            FOR i := 1 TO 10 DO
                GVL_1.Condition_Cr_A[condNo].Row[i].Enable   := GVL.HMI_A_CondEditRowEnable[i];
                GVL_1.Condition_Cr_A[condNo].Row[i].Source   := GVL.HMI_A_CondEditSource[i];
                GVL_1.Condition_Cr_A[condNo].Row[i].Index    := GVL.HMI_A_CondEditIndex[i];
                GVL_1.Condition_Cr_A[condNo].Row[i].Operator := GVL.HMI_A_CondEditOperator[i];
                GVL_1.Condition_Cr_A[condNo].Row[i].SetValue := GVL.HMI_A_CondEditSetValue[i];
                GVL_1.Condition_Cr_A[condNo].Row[i].LinkNext := GVL.HMI_A_CondEditLinkNext[i];
                //GVL_1.Condition_Cr_A[condNo].Row[i].Note     := GVL.HMI_A_CondEditNote[i];
            END_FOR;
        END_IF;

        GVL.HMI_A_CondCmdReq := 0;


    3: // Clear condition
        condNo := GVL.HMI_A_CondSelectedNo;

        IF (condNo >= 1) AND (condNo <= 100) THEN
            GVL_1.Condition_Cr_A[condNo].Enable := FALSE;
            GVL_1.Condition_Cr_A[condNo].Name := '';

            FOR i := 1 TO 10 DO
                GVL_1.Condition_Cr_A[condNo].Row[i].Enable := FALSE;
                GVL_1.Condition_Cr_A[condNo].Row[i].Source := 0;
                GVL_1.Condition_Cr_A[condNo].Row[i].Index := 0;
                GVL_1.Condition_Cr_A[condNo].Row[i].Operator := 0;
                GVL_1.Condition_Cr_A[condNo].Row[i].SetValue := 0;
                GVL_1.Condition_Cr_A[condNo].Row[i].LinkNext := 0;
                //GVL_1.Condition_Cr_A[condNo].Row[i].Note := '';
            END_FOR;
        END_IF;

        GVL.HMI_A_CondCmdReq := 0;


    4: // Copy
        condNo := GVL.HMI_A_CondSelectedNo;

        IF (condNo >= 1) AND (condNo <= 100) THEN
            GVL.HMI_A_CondCopied := GVL_1.Condition_Cr_A[condNo];
        END_IF;

        GVL.HMI_A_CondCmdReq := 0;


    5: // Paste
        condNo := GVL.HMI_A_CondEditNo;

        IF (condNo >= 1) AND (condNo <= 100) THEN
            GVL_1.Condition_Cr_A[condNo] := GVL.HMI_A_CondCopied;
        END_IF;

        GVL.HMI_A_CondCmdReq := 1; // Load lại lên Edit


    6: // Delete Row
        rowNo := GVL.HMI_A_CondSelectedNo;

        IF (rowNo >= 1) AND (rowNo <= 10) THEN
            FOR i := rowNo TO 9 DO
                GVL.HMI_A_CondEditRowEnable[i] := GVL.HMI_A_CondEditRowEnable[i + 1];
                GVL.HMI_A_CondEditSource[i]    := GVL.HMI_A_CondEditSource[i + 1];
                GVL.HMI_A_CondEditIndex[i]     := GVL.HMI_A_CondEditIndex[i + 1];
                GVL.HMI_A_CondEditOperator[i]  := GVL.HMI_A_CondEditOperator[i + 1];
                GVL.HMI_A_CondEditSetValue[i]  := GVL.HMI_A_CondEditSetValue[i + 1];
                GVL.HMI_A_CondEditLinkNext[i]  := GVL.HMI_A_CondEditLinkNext[i + 1];
                GVL.HMI_A_CondEditNote[i]      := GVL.HMI_A_CondEditNote[i + 1];
            END_FOR;

            GVL.HMI_A_CondEditRowEnable[10] := FALSE;
            GVL.HMI_A_CondEditSource[10] := 0;
            GVL.HMI_A_CondEditIndex[10] := 0;
            GVL.HMI_A_CondEditOperator[10] := 0;
            GVL.HMI_A_CondEditSetValue[10] := 0;
            GVL.HMI_A_CondEditLinkNext[10] := 0;
            GVL.HMI_A_CondEditNote[10] := '';
        END_IF;

        GVL.HMI_A_CondCmdReq := 0;


    7: // Insert Row
        rowNo := GVL.HMI_A_CondSelectedNo;

        IF (rowNo >= 1) AND (rowNo <= 10) THEN
            FOR i := 10 TO rowNo + 1 BY -1 DO
                GVL.HMI_A_CondEditRowEnable[i] := GVL.HMI_A_CondEditRowEnable[i - 1];
                GVL.HMI_A_CondEditSource[i]    := GVL.HMI_A_CondEditSource[i - 1];
                GVL.HMI_A_CondEditIndex[i]     := GVL.HMI_A_CondEditIndex[i - 1];
                GVL.HMI_A_CondEditOperator[i]  := GVL.HMI_A_CondEditOperator[i - 1];
                GVL.HMI_A_CondEditSetValue[i]  := GVL.HMI_A_CondEditSetValue[i - 1];
                GVL.HMI_A_CondEditLinkNext[i]  := GVL.HMI_A_CondEditLinkNext[i - 1];
                GVL.HMI_A_CondEditNote[i]      := GVL.HMI_A_CondEditNote[i - 1];
            END_FOR;

            GVL.HMI_A_CondEditRowEnable[rowNo] := FALSE;
            GVL.HMI_A_CondEditSource[rowNo] := 0;
            GVL.HMI_A_CondEditIndex[rowNo] := 0;
            GVL.HMI_A_CondEditOperator[rowNo] := 0;
            GVL.HMI_A_CondEditSetValue[rowNo] := 0;
            GVL.HMI_A_CondEditLinkNext[rowNo] := 0;
            GVL.HMI_A_CondEditNote[rowNo] := '';
        END_IF;

        GVL.HMI_A_CondCmdReq := 0;

END_CASE;


// PRG_A_ConditionScan -- PRG quét realtime kết quả Condition
FOR i := 1 TO 100 DO
    GVL_1.Condition_Cr_A[i].Result := F_EvalCondition_A(i);
END_FOR;

//====================================================
// CONDITION EDIT MONITOR
// Khi bật Monitor, hiển thị ActualValue / RowResult / FinalResult
// theo vùng đang edit, kể cả chưa Save
//====================================================

IF GVL.HMI_A_CondMonitorEnable THEN

    firstRow := TRUE;
    finalResult := FALSE;

    FOR i := 1 TO 10 DO

        IF GVL.HMI_A_CondEditRowEnable[i] THEN

            rowResult := F_EvalCondRowFromEdit_A(i);

            GVL.HMI_A_CondMonRowResult[i] := rowResult;

            IF firstRow THEN
                finalResult := rowResult;
                firstRow := FALSE;
            ELSE
                CASE GVL.HMI_A_CondEditLinkNext[i - 1] OF
                    1: finalResult := finalResult AND rowResult;
                    2: finalResult := finalResult OR rowResult;
                ELSE
                    finalResult := finalResult AND rowResult;
                END_CASE;
            END_IF;

        ELSE
            GVL.HMI_A_CondMonActualValue[i] := 0;
            GVL.HMI_A_CondMonRowResult[i] := FALSE;
        END_IF;

    END_FOR;

    GVL.HMI_A_CondMonFinalResult := finalResult;

ELSE
    GVL.HMI_A_CondMonFinalResult := FALSE;

    FOR i := 1 TO 10 DO
        GVL.HMI_A_CondMonActualValue[i] := 0;
        GVL.HMI_A_CondMonRowResult[i] := FALSE;
    END_FOR;
END_IF;
END_ACTION

ACTION ACT_HMI_A_Vision_Tracking_Config:
//=============================================================================
// ACT_HMI_A_Vision_Tracking_Config
//-----------------------------------------------------------------------------
// HMI editor cho Vision Tracking Source Robot A.
// Pattern giống Sensor Source:
// Index -> Edit Struct -> Load / Save.
//=============================================================================


//=============================================================================
// 01. KIỂM TRA INDEX
//=============================================================================
IF GVL.g_uiHMIVisionSourceIndexA = 0
OR GVL.g_uiHMIVisionSourceIndexA > GVL.C_MAX_VISION_CHANNELS THEN
    GVL.g_uiHMIVisionSourceIndexA := 1;
END_IF;


//=============================================================================
// 02. LOAD SOURCE -> HMI BUFFER
//=============================================================================
IF GVL.g_xHMILoadVisionSourceA THEN

    GVL.g_stHMIVisionSourceA :=
        GVL.g_aVisionTrackingSourceConfigA[
            GVL.g_uiHMIVisionSourceIndexA
        ];

    GVL.g_xHMILoadVisionSourceA := FALSE;

END_IF;


//=============================================================================
// 03. SAVE HMI BUFFER -> SOURCE
//=============================================================================
IF GVL.g_xHMISaveVisionSourceA THEN

    GVL.g_aVisionTrackingSourceConfigA[
        GVL.g_uiHMIVisionSourceIndexA
    ] := GVL.g_stHMIVisionSourceA;

    GVL.g_xHMISaveVisionSourceA := FALSE;

    // Yêu cầu lưu toàn bộ Vision Source xuống file.
    GVL.g_xHMISaveAllVisionSourceA := TRUE;

END_IF;
END_ACTION

ACTION ACT_HMI_B_ConditionEditor:
//====================================================
// PRG_HMI_A_ConditionEditor
// Hiển thị danh sách condition + xử lý Load/Save/Edit
//====================================================

// Scroll danh sách condition
IF GVL.HMI_B_CondCmd_Up THEN
    GVL.HMI_B_CondCmd_Up := FALSE;
    IF GVL.HMI_B_CondViewStart > 1 THEN
        GVL.HMI_B_CondViewStart := GVL.HMI_B_CondViewStart - 1;
    END_IF;
END_IF;

IF GVL.HMI_B_CondCmd_Down THEN
    GVL.HMI_B_CondCmd_Down := FALSE;
    IF GVL.HMI_B_CondViewStart < 91 THEN
        GVL.HMI_B_CondViewStart := GVL.HMI_B_CondViewStart + 1;
    END_IF;
END_IF;

IF GVL.HMI_B_CondCmd_PageUp THEN
    GVL.HMI_B_CondCmd_PageUp := FALSE;
    GVL.HMI_B_CondViewStart := GVL.HMI_B_CondViewStart - 10;
    IF GVL.HMI_B_CondViewStart < 1 THEN
        GVL.HMI_B_CondViewStart := 1;
    END_IF;
END_IF;

IF GVL.HMI_B_CondCmd_PageDown THEN
    GVL.HMI_B_CondCmd_PageDown := FALSE;
    GVL.HMI_B_CondViewStart := GVL.HMI_B_CondViewStart + 10;
    IF GVL.HMI_B_CondViewStart > 91 THEN
        GVL.HMI_B_CondViewStart := 91;
    END_IF;
END_IF;

IF GVL.HMI_B_CondCmd_GoTop THEN
    GVL.HMI_B_CondCmd_GoTop := FALSE;
    GVL.HMI_B_CondViewStart := 1;
END_IF;

IF GVL.HMI_B_CondCmd_GoBot THEN
    GVL.HMI_B_CondCmd_GoBot := FALSE;
    GVL.HMI_B_CondViewStart := 91;
END_IF;


//====================================================
// Row Select
//====================================================

FOR i := 1 TO 10 DO
    IF (GVL.HMI_B_CondSelectedCmd = i) THEN
		GVL.HMI_B_CondRowSelect[i] := TRUE;
		GVL.HMI_B_CondSelectedNo := i + GVL.HMI_B_CondViewStart - 1;
		//GVL.HMI_B_EditStepNo   := GVL.HMI_B_SelectedStepNo;
	ELSE
		GVL.HMI_B_CondRowSelect[i] := FALSE;
    END_IF;
END_FOR;

// FOR i := 1 TO 10 DO
//     IF GVL.HMI_B_CondRowSelect[i] THEN
//         GVL.HMI_B_CondRowSelect[i] := FALSE;
//         condNo := GVL.HMI_B_CondViewNo[i];
// 
//         IF (condNo >= 1) AND (condNo <= 100) THEN
//             GVL.HMI_B_CondSelectedNo := condNo;
//             GVL.HMI_B_CondCmdReq := 1; // Load
//         END_IF;
//     END_IF;
// END_FOR;


//====================================================
// Update View 10 dòng condition
//====================================================
FOR i := 1 TO 10 DO
    condNo := GVL.HMI_B_CondViewStart + i - 1;

    IF (condNo >= 1) AND (condNo <= 100) THEN
        GVL.HMI_B_CondViewNo[i]     := condNo;
        GVL.HMI_B_CondViewName[i]   := GVL_1.Condition_Cr_B[condNo].Name;
        GVL.HMI_B_CondViewEnable[i] := GVL_1.Condition_Cr_B[condNo].Enable;
        GVL.HMI_B_CondViewResult[i] := GVL_1.Condition_Cr_B[condNo].Result;
    ELSE
        GVL.HMI_B_CondViewNo[i]     := 0;
        GVL.HMI_B_CondViewName[i]   := '';
        GVL.HMI_B_CondViewEnable[i] := FALSE;
        GVL.HMI_B_CondViewResult[i] := FALSE;
    END_IF;
END_FOR;


//====================================================
// Command Load / Save / Clear / Copy / Paste
//====================================================
CASE GVL.HMI_B_CondCmdReq OF

    1: // Load condition vào vùng Edit
        condNo := GVL.HMI_B_CondSelectedNo;

        IF (condNo >= 1) AND (condNo <= 100) THEN
            GVL.HMI_B_CondEditNo := condNo;
            GVL.HMI_B_CondEditName := GVL_1.Condition_Cr_B[condNo].Name;
            GVL.HMI_B_CondEditEnable := GVL_1.Condition_Cr_B[condNo].Enable;

            FOR i := 1 TO 10 DO
                GVL.HMI_B_CondEditRowEnable[i] := GVL_1.Condition_Cr_B[condNo].Row[i].Enable;
                GVL.HMI_B_CondEditSource[i]    := GVL_1.Condition_Cr_B[condNo].Row[i].Source;
                GVL.HMI_B_CondEditIndex[i]     := GVL_1.Condition_Cr_B[condNo].Row[i].Index;
                GVL.HMI_B_CondEditOperator[i]  := GVL_1.Condition_Cr_B[condNo].Row[i].Operator;
                GVL.HMI_B_CondEditSetValue[i]  := GVL_1.Condition_Cr_B[condNo].Row[i].SetValue;
                GVL.HMI_B_CondEditLinkNext[i]  := GVL_1.Condition_Cr_B[condNo].Row[i].LinkNext;
                //GVL.HMI_B_CondEditNote[i]      := GVL_1.Condition_Cr_B[condNo].Row[i].Note;
            END_FOR;
        END_IF;

        GVL.HMI_B_CondCmdReq := 0;


    2: // Save vùng Edit về bảng thật
        condNo := GVL.HMI_B_CondSelectedNo;

        IF (condNo >= 1) AND (condNo <= 100) THEN
            GVL_1.Condition_Cr_B[condNo].Name := GVL.HMI_B_CondEditName;
            GVL_1.Condition_Cr_B[condNo].Enable := GVL.HMI_B_CondEditEnable;

            FOR i := 1 TO 10 DO
                GVL_1.Condition_Cr_B[condNo].Row[i].Enable   := GVL.HMI_B_CondEditRowEnable[i];
                GVL_1.Condition_Cr_B[condNo].Row[i].Source   := GVL.HMI_B_CondEditSource[i];
                GVL_1.Condition_Cr_B[condNo].Row[i].Index    := GVL.HMI_B_CondEditIndex[i];
                GVL_1.Condition_Cr_B[condNo].Row[i].Operator := GVL.HMI_B_CondEditOperator[i];
                GVL_1.Condition_Cr_B[condNo].Row[i].SetValue := GVL.HMI_B_CondEditSetValue[i];
                GVL_1.Condition_Cr_B[condNo].Row[i].LinkNext := GVL.HMI_B_CondEditLinkNext[i];
                //GVL_1.Condition_Cr_B[condNo].Row[i].Note     := GVL.HMI_B_CondEditNote[i];
            END_FOR;
        END_IF;

        GVL.HMI_B_CondCmdReq := 0;


    3: // Clear condition
        condNo := GVL.HMI_B_CondSelectedNo;

        IF (condNo >= 1) AND (condNo <= 100) THEN
            GVL_1.Condition_Cr_B[condNo].Enable := FALSE;
            GVL_1.Condition_Cr_B[condNo].Name := '';

            FOR i := 1 TO 10 DO
                GVL_1.Condition_Cr_B[condNo].Row[i].Enable := FALSE;
                GVL_1.Condition_Cr_B[condNo].Row[i].Source := 0;
                GVL_1.Condition_Cr_B[condNo].Row[i].Index := 0;
                GVL_1.Condition_Cr_B[condNo].Row[i].Operator := 0;
                GVL_1.Condition_Cr_B[condNo].Row[i].SetValue := 0;
                GVL_1.Condition_Cr_B[condNo].Row[i].LinkNext := 0;
                //GVL_1.Condition_Cr_B[condNo].Row[i].Note := '';
            END_FOR;
        END_IF;

        GVL.HMI_B_CondCmdReq := 0;


    4: // Copy
        condNo := GVL.HMI_B_CondSelectedNo;

        IF (condNo >= 1) AND (condNo <= 100) THEN
            GVL.HMI_B_CondCopied := GVL_1.Condition_Cr_B[condNo];
        END_IF;

        GVL.HMI_B_CondCmdReq := 0;


    5: // Paste
        condNo := GVL.HMI_B_CondEditNo;

        IF (condNo >= 1) AND (condNo <= 100) THEN
            GVL_1.Condition_Cr_B[condNo] := GVL.HMI_B_CondCopied;
        END_IF;

        GVL.HMI_B_CondCmdReq := 1; // Load lại lên Edit


    6: // Delete Row
        rowNo := GVL.HMI_B_CondSelectedNo;

        IF (rowNo >= 1) AND (rowNo <= 10) THEN
            FOR i := rowNo TO 9 DO
                GVL.HMI_B_CondEditRowEnable[i] := GVL.HMI_B_CondEditRowEnable[i + 1];
                GVL.HMI_B_CondEditSource[i]    := GVL.HMI_B_CondEditSource[i + 1];
                GVL.HMI_B_CondEditIndex[i]     := GVL.HMI_B_CondEditIndex[i + 1];
                GVL.HMI_B_CondEditOperator[i]  := GVL.HMI_B_CondEditOperator[i + 1];
                GVL.HMI_B_CondEditSetValue[i]  := GVL.HMI_B_CondEditSetValue[i + 1];
                GVL.HMI_B_CondEditLinkNext[i]  := GVL.HMI_B_CondEditLinkNext[i + 1];
                GVL.HMI_B_CondEditNote[i]      := GVL.HMI_B_CondEditNote[i + 1];
            END_FOR;

            GVL.HMI_B_CondEditRowEnable[10] := FALSE;
            GVL.HMI_B_CondEditSource[10] := 0;
            GVL.HMI_B_CondEditIndex[10] := 0;
            GVL.HMI_B_CondEditOperator[10] := 0;
            GVL.HMI_B_CondEditSetValue[10] := 0;
            GVL.HMI_B_CondEditLinkNext[10] := 0;
            GVL.HMI_B_CondEditNote[10] := '';
        END_IF;

        GVL.HMI_B_CondCmdReq := 0;


    7: // Insert Row
        rowNo := GVL.HMI_B_CondSelectedNo;

        IF (rowNo >= 1) AND (rowNo <= 10) THEN
            FOR i := 10 TO rowNo + 1 BY -1 DO
                GVL.HMI_B_CondEditRowEnable[i] := GVL.HMI_B_CondEditRowEnable[i - 1];
                GVL.HMI_B_CondEditSource[i]    := GVL.HMI_B_CondEditSource[i - 1];
                GVL.HMI_B_CondEditIndex[i]     := GVL.HMI_B_CondEditIndex[i - 1];
                GVL.HMI_B_CondEditOperator[i]  := GVL.HMI_B_CondEditOperator[i - 1];
                GVL.HMI_B_CondEditSetValue[i]  := GVL.HMI_B_CondEditSetValue[i - 1];
                GVL.HMI_B_CondEditLinkNext[i]  := GVL.HMI_B_CondEditLinkNext[i - 1];
                GVL.HMI_B_CondEditNote[i]      := GVL.HMI_B_CondEditNote[i - 1];
            END_FOR;

            GVL.HMI_B_CondEditRowEnable[rowNo] := FALSE;
            GVL.HMI_B_CondEditSource[rowNo] := 0;
            GVL.HMI_B_CondEditIndex[rowNo] := 0;
            GVL.HMI_B_CondEditOperator[rowNo] := 0;
            GVL.HMI_B_CondEditSetValue[rowNo] := 0;
            GVL.HMI_B_CondEditLinkNext[rowNo] := 0;
            GVL.HMI_B_CondEditNote[rowNo] := '';
        END_IF;

        GVL.HMI_B_CondCmdReq := 0;

END_CASE;


// PRG_A_ConditionScan -- PRG quét realtime kết quả Condition
FOR i := 1 TO 100 DO
    GVL_1.Condition_Cr_B[i].Result := F_EvalCondition_B(i);
END_FOR;

//====================================================
// CONDITION EDIT MONITOR
// Khi bật Monitor, hiển thị ActualValue / RowResult / FinalResult
// theo vùng đang edit, kể cả chưa Save
//====================================================

IF GVL.HMI_B_CondMonitorEnable THEN

    firstRow := TRUE;
    finalResult := FALSE;

    FOR i := 1 TO 10 DO

        IF GVL.HMI_B_CondEditRowEnable[i] THEN

            rowResult := F_EvalCondRowFromEdit_B(i);

            GVL.HMI_B_CondMonRowResult[i] := rowResult;

            IF firstRow THEN
                finalResult := rowResult;
                firstRow := FALSE;
            ELSE
                CASE GVL.HMI_B_CondEditLinkNext[i - 1] OF
                    1: finalResult := finalResult AND rowResult;
                    2: finalResult := finalResult OR rowResult;
                ELSE
                    finalResult := finalResult AND rowResult;
                END_CASE;
            END_IF;

        ELSE
            GVL.HMI_B_CondMonActualValue[i] := 0;
            GVL.HMI_B_CondMonRowResult[i] := FALSE;
        END_IF;

    END_FOR;

    GVL.HMI_B_CondMonFinalResult := finalResult;

ELSE
    GVL.HMI_B_CondMonFinalResult := FALSE;

    FOR i := 1 TO 10 DO
        GVL.HMI_B_CondMonActualValue[i] := 0;
        GVL.HMI_B_CondMonRowResult[i] := FALSE;
    END_FOR;
END_IF;
END_ACTION

ACTION ACT_HMI_B_Vision_Tracking_Config:
// CREATE ACTION under POU_HMI_CONTROL_ROBOT: ACT_HMI_B_Vision_Tracking_Config

//=============================================================================
// ACT_HMI_B_Vision_Tracking_Config
//-----------------------------------------------------------------------------
// HMI editor cho Vision Tracking Source Robot B.
// Pattern giống Sensor Source:
// Index -> Edit Struct -> Load / Save.
//=============================================================================


//=============================================================================
// 01. KIỂM TRA INDEX
//=============================================================================
IF GVL.g_uiHMIVisionSourceIndexB = 0
OR GVL.g_uiHMIVisionSourceIndexB > GVL.C_MAX_VISION_CHANNELS THEN
    GVL.g_uiHMIVisionSourceIndexB := 1;
END_IF;


//=============================================================================
// 02. LOAD SOURCE -> HMI BUFFER
//=============================================================================
IF GVL.g_xHMILoadVisionSourceB THEN

    GVL.g_stHMIVisionSourceB :=
        GVL.g_aVisionTrackingSourceConfigB[
            GVL.g_uiHMIVisionSourceIndexB
        ];

    GVL.g_xHMILoadVisionSourceB := FALSE;

END_IF;


//=============================================================================
// 03. SAVE HMI BUFFER -> SOURCE
//=============================================================================
IF GVL.g_xHMISaveVisionSourceB THEN

    GVL.g_aVisionTrackingSourceConfigB[
        GVL.g_uiHMIVisionSourceIndexB
    ] := GVL.g_stHMIVisionSourceB;

    GVL.g_xHMISaveVisionSourceB := FALSE;

    // Yêu cầu lưu toàn bộ Vision Source xuống file.
    GVL.g_xHMISaveAllVisionSourceB := TRUE;

END_IF;
END_ACTION

ACTION ACT_HMI_Recipe_Config:
//=============================================================================
// TRACKING RECIPE HMI LOAD / SAVE
//=============================================================================

//=============================================================================
// 03. KHỞI TẠO INDEX MẶC ĐỊNH
//=============================================================================
IF GVL.g_uiHMITrackingRecipeIndexA = 0 OR GVL.g_uiHMITrackingRecipeIndexA > GVL.C_MAX_TRACK_RECIPES THEN
    GVL.g_uiHMITrackingRecipeIndexA := 1;
END_IF;

//-----------------------------------------------------------------------------
// LOAD
//-----------------------------------------------------------------------------
IF GVL.g_xHMILoadTrackingRecipeA THEN

    IF (GVL.g_uiHMITrackingRecipeIndexA >= 1)
    AND (GVL.g_uiHMITrackingRecipeIndexA <= GVL.C_MAX_TRACK_RECIPES) THEN

        GVL.g_stHMITrackingRecipeA :=
            GVL.g_aMultiTrackRecipeA[GVL.g_uiHMITrackingRecipeIndexA];

    END_IF;

    GVL.g_xHMILoadTrackingRecipeA := FALSE;

END_IF;


//-----------------------------------------------------------------------------
// SAVE
//-----------------------------------------------------------------------------
IF GVL.g_xHMISaveTrackingRecipeA THEN

    IF (GVL.g_uiHMITrackingRecipeIndexA >= 1)
    AND (GVL.g_uiHMITrackingRecipeIndexA <= GVL.C_MAX_TRACK_RECIPES) THEN

        GVL.g_aMultiTrackRecipeA[GVL.g_uiHMITrackingRecipeIndexA] :=
            GVL.g_stHMITrackingRecipeA;

    END_IF;

    GVL.g_xHMISaveTrackingRecipeA := FALSE;
	GVL.g_xHMISaveTrackingRecipeA_All := TRUE;

END_IF;
END_ACTION

ACTION ACT_HMI_Recipe_Config_B:
// CREATE ACTION under POU_HMI_CONTROL_ROBOT: ACT_HMI_Recipe_Config_B

//=============================================================================
// TRACKING RECIPE HMI LOAD / SAVE
//=============================================================================

//=============================================================================
// 03. KHỞI TẠO INDEX MẶC ĐỊNH
//=============================================================================
IF GVL.g_uiHMITrackingRecipeIndexB = 0 OR GVL.g_uiHMITrackingRecipeIndexB > GVL.C_MAX_TRACK_RECIPES THEN
    GVL.g_uiHMITrackingRecipeIndexB := 1;
END_IF;

//-----------------------------------------------------------------------------
// LOAD
//-----------------------------------------------------------------------------
IF GVL.g_xHMILoadTrackingRecipeB THEN

    IF (GVL.g_uiHMITrackingRecipeIndexB >= 1)
    AND (GVL.g_uiHMITrackingRecipeIndexB <= GVL.C_MAX_TRACK_RECIPES) THEN

        GVL.g_stHMITrackingRecipeB :=
            GVL.g_aMultiTrackRecipeB[GVL.g_uiHMITrackingRecipeIndexB];

    END_IF;

    GVL.g_xHMILoadTrackingRecipeB := FALSE;

END_IF;


//-----------------------------------------------------------------------------
// SAVE
//-----------------------------------------------------------------------------
IF GVL.g_xHMISaveTrackingRecipeB THEN

    IF (GVL.g_uiHMITrackingRecipeIndexB >= 1)
    AND (GVL.g_uiHMITrackingRecipeIndexB <= GVL.C_MAX_TRACK_RECIPES) THEN

        GVL.g_aMultiTrackRecipeB[GVL.g_uiHMITrackingRecipeIndexB] :=
            GVL.g_stHMITrackingRecipeB;

    END_IF;

    GVL.g_xHMISaveTrackingRecipeB := FALSE;
	GVL.g_xHMISaveTrackingRecipeB_All := TRUE;

END_IF;
END_ACTION

ACTION ACT_HMI_SensorSource_Config_B:
// CREATE ACTION under POU_HMI_CONTROL_ROBOT: ACT_HMI_SensorSource_Config_B

//=============================================================================
// SENSOR SOURCE HMI LOAD / SAVE
//=============================================================================

//=============================================================================
// 03. KHỞI TẠO INDEX MẶC ĐỊNH
//=============================================================================
IF GVL.g_uiHMISensorSourceIndexB = 0 OR GVL.g_uiHMISensorSourceIndexB > GVL.C_MAX_SENSOR_SOURCES THEN
    GVL.g_uiHMISensorSourceIndexB := 1;
END_IF;



//-----------------------------------------------------------------------------
// LOAD
//-----------------------------------------------------------------------------
IF GVL.g_xHMILoadSensorSourceB THEN

    IF (GVL.g_uiHMISensorSourceIndexB >= 1)
    AND (GVL.g_uiHMISensorSourceIndexB <= GVL.C_MAX_SENSOR_SOURCES) THEN

        GVL.g_stHMISensorSourceB :=
            GVL.g_aSensorSourceConfigB[GVL.g_uiHMISensorSourceIndexB];

    END_IF;

    GVL.g_xHMILoadSensorSourceB := FALSE;

END_IF;


//-----------------------------------------------------------------------------
// SAVE
//-----------------------------------------------------------------------------
IF GVL.g_xHMISaveSensorSourceB THEN

    IF (GVL.g_uiHMISensorSourceIndexB >= 1)
    AND (GVL.g_uiHMISensorSourceIndexB <= GVL.C_MAX_SENSOR_SOURCES) THEN

        GVL.g_aSensorSourceConfigB[GVL.g_uiHMISensorSourceIndexB] :=
            GVL.g_stHMISensorSourceB;

    END_IF;

    GVL.g_xHMISaveSensorSourceB := FALSE;
	GVL.g_xHMISaveSensorSourceB_All := TRUE;

END_IF;
END_ACTION

ACTION ACT_HMI_SensorSource_Config:
//=============================================================================
// SENSOR SOURCE HMI LOAD / SAVE
//=============================================================================

//=============================================================================
// 03. KHỞI TẠO INDEX MẶC ĐỊNH
//=============================================================================
IF GVL.g_uiHMISensorSourceIndexA = 0 OR GVL.g_uiHMISensorSourceIndexA > GVL.C_MAX_SENSOR_SOURCES THEN
    GVL.g_uiHMISensorSourceIndexA := 1;
END_IF;



//-----------------------------------------------------------------------------
// LOAD
//-----------------------------------------------------------------------------
IF GVL.g_xHMILoadSensorSourceA THEN

    IF (GVL.g_uiHMISensorSourceIndexA >= 1)
    AND (GVL.g_uiHMISensorSourceIndexA <= GVL.C_MAX_SENSOR_SOURCES) THEN

        GVL.g_stHMISensorSourceA :=
            GVL.g_aSensorSourceConfigA[GVL.g_uiHMISensorSourceIndexA];

    END_IF;

    GVL.g_xHMILoadSensorSourceA := FALSE;

END_IF;


//-----------------------------------------------------------------------------
// SAVE
//-----------------------------------------------------------------------------
IF GVL.g_xHMISaveSensorSourceA THEN

    IF (GVL.g_uiHMISensorSourceIndexA >= 1)
    AND (GVL.g_uiHMISensorSourceIndexA <= GVL.C_MAX_SENSOR_SOURCES) THEN

        GVL.g_aSensorSourceConfigA[GVL.g_uiHMISensorSourceIndexA] :=
            GVL.g_stHMISensorSourceA;

    END_IF;

    GVL.g_xHMISaveSensorSourceA := FALSE;
	GVL.g_xHMISaveSensorSourceA_All := TRUE;

END_IF;
END_ACTION

ACTION ACT_HMIToolConfigEditor_A:
//=============================================================================
// PROGRAM: PRG_HMIToolConfigEditor_A
//-----------------------------------------------------------------------------
// Quản lý trang HMI cấu hình nhiều Tool cho Robot A.
//
// NGUYÊN TẮC:
// 1. HMI chỉnh EditData, không chỉnh trực tiếp g_aToolConfigA.
// 2. Load sao chép ToolConfig vào EditData.
// 3. Save kiểm tra dữ liệu rồi mới ghi về ToolConfig.
// 4. Cancel khôi phục dữ liệu từ OriginalData.
// 5. Save luôn ghi theo LoadedIndex để tránh ghi nhầm Tool.
//=============================================================================


//=============================================================================
// 01. BẮT CẠNH LỆNH HMI
//=============================================================================
GVL.g_rtHMIToolLoadA(CLK := GVL.g_stHMIToolEditorA.LoadCommand);

GVL.g_rtHMIToolSaveA(CLK := GVL.g_stHMIToolEditorA.SaveCommand);

GVL.g_rtHMIToolCancelA(CLK := GVL.g_stHMIToolEditorA.CancelCommand);


//=============================================================================
// 02. OUTPUT DẠNG XUNG
//-----------------------------------------------------------------------------
// LoadDone và SaveDone chỉ TRUE trong một vòng quét.
//=============================================================================
GVL.g_stHMIToolEditorA.LoadDone := FALSE;
GVL.g_stHMIToolEditorA.SaveDone := FALSE;
GVL.g_stHMIToolEditorA.Busy := FALSE;


//=============================================================================
// 03. KHỞI TẠO INDEX MẶC ĐỊNH
//=============================================================================
IF GVL.g_stHMIToolEditorA.SelectedIndex = 0 THEN
    GVL.g_stHMIToolEditorA.SelectedIndex := 1;
END_IF;


//=============================================================================
// 04. TỰ ĐỘNG LOAD KHI ĐỔI TOOL
//-----------------------------------------------------------------------------
// Chỉ tự động Load khi dữ liệu hiện tại chưa bị chỉnh sửa.
// Nếu DataChanged = TRUE thì giữ dữ liệu hiện tại để tránh mất dữ liệu.
//=============================================================================
IF GVL.g_stHMIToolEditorA.SelectedIndex <> GVL.g_uiHMIToolSelectedIndexOldA THEN

    IF GVL.g_stHMIToolEditorA.DataChanged THEN

        // Không cho đổi Tool khi dữ liệu hiện tại chưa được Save hoặc Cancel.
        GVL.g_stHMIToolEditorA.SelectedIndex := GVL.g_uiHMIToolSelectedIndexOldA;

        GVL.g_stHMIToolEditorA.Error := TRUE;
        GVL.g_stHMIToolEditorA.ErrorID := 1101;

    ELSIF GVL.g_stHMIToolEditorA.SelectedIndex >= 1 AND GVL.g_stHMIToolEditorA.SelectedIndex <= GVL.C_MAX_TOOLS THEN

        // Sao chép cấu hình Tool được chọn vào vùng chỉnh sửa.
        GVL.g_stHMIToolEditorA.EditData := GVL.g_aToolConfigA[GVL.g_stHMIToolEditorA.SelectedIndex];

        // Lưu bản gốc để phục vụ Cancel.
        GVL.g_stHMIToolEditorA.OriginalData := GVL.g_aToolConfigA[GVL.g_stHMIToolEditorA.SelectedIndex];

        GVL.g_stHMIToolEditorA.LoadedIndex := GVL.g_stHMIToolEditorA.SelectedIndex;

        GVL.g_uiHMIToolSelectedIndexOldA := GVL.g_stHMIToolEditorA.SelectedIndex;

        GVL.g_stHMIToolEditorA.DataChanged := FALSE;
        GVL.g_stHMIToolEditorA.Error := FALSE;
        GVL.g_stHMIToolEditorA.ErrorID := 0;
        GVL.g_stHMIToolEditorA.LoadDone := TRUE;

    ELSE

        // Index Tool ngoài phạm vi.
        GVL.g_stHMIToolEditorA.Error := TRUE;
        GVL.g_stHMIToolEditorA.ErrorID := 1102;

    END_IF;

END_IF;


//=============================================================================
// 05. LOAD THỦ CÔNG
//=============================================================================
IF GVL.g_rtHMIToolLoadA.Q THEN

    GVL.g_stHMIToolEditorA.Busy := TRUE;
    GVL.g_stHMIToolEditorA.Error := FALSE;
    GVL.g_stHMIToolEditorA.ErrorID := 0;

    IF GVL.g_stHMIToolEditorA.SelectedIndex >= 1
    AND GVL.g_stHMIToolEditorA.SelectedIndex <= GVL.C_MAX_TOOLS THEN

        GVL.g_stHMIToolEditorA.EditData := GVL.g_aToolConfigA[GVL.g_stHMIToolEditorA.SelectedIndex];

        GVL.g_stHMIToolEditorA.OriginalData := GVL.g_aToolConfigA[GVL.g_stHMIToolEditorA.SelectedIndex];

        GVL.g_stHMIToolEditorA.LoadedIndex := GVL.g_stHMIToolEditorA.SelectedIndex;

        GVL.g_uiHMIToolSelectedIndexOldA := GVL.g_stHMIToolEditorA.SelectedIndex;

        GVL.g_stHMIToolEditorA.DataChanged := FALSE;
        GVL.g_stHMIToolEditorA.LoadDone := TRUE;

    ELSE

        GVL.g_stHMIToolEditorA.Error := TRUE;
        GVL.g_stHMIToolEditorA.ErrorID := 1102;

    END_IF;
	
	GVL.g_stHMIToolEditorA.LoadCommand := FALSE;

END_IF;


// //=============================================================================
// // 06. CANCEL THAY ĐỔI
// //-----------------------------------------------------------------------------
// // Khôi phục EditData về bản dữ liệu đã Load gần nhất.
// //=============================================================================
// IF GVL.g_rtHMIToolCancelA.Q THEN
// 
//     GVL.g_stHMIToolEditorA.Busy := TRUE;
//     GVL.g_stHMIToolEditorA.Error := FALSE;
//     GVL.g_stHMIToolEditorA.ErrorID := 0;
// 
//     IF GVL.g_stHMIToolEditorA.LoadedIndex >= 1
//     AND GVL.g_stHMIToolEditorA.LoadedIndex <= GVL.C_MAX_TOOLS THEN
// 
//         GVL.g_stHMIToolEditorA.EditData := GVL.g_stHMIToolEditorA.OriginalData;
// 
//         GVL.g_stHMIToolEditorA.DataChanged := FALSE;
//         GVL.g_stHMIToolEditorA.LoadDone := TRUE;
// 
//     ELSE
// 
//         GVL.g_stHMIToolEditorA.Error := TRUE;
//         GVL.g_stHMIToolEditorA.ErrorID := 1103;
// 
//     END_IF;
// 
// END_IF;


//=============================================================================
// 07. SAVE CẤU HÌNH TOOL
//=============================================================================
IF GVL.g_rtHMIToolSaveA.Q THEN

    GVL.g_stHMIToolEditorA.Busy := TRUE;
    GVL.g_stHMIToolEditorA.Error := FALSE;
    GVL.g_stHMIToolEditorA.ErrorID := 0;
    GVL.g_xHMIToolDuplicateIDA := FALSE;

    //-------------------------------------------------------------------------
    // Kiểm tra ToolID có trùng với Tool khác hay không.
    //-------------------------------------------------------------------------
    FOR GVL.g_uiHMIToolCheckIndexA := 1 TO GVL.C_MAX_TOOLS DO

        IF GVL.g_uiHMIToolCheckIndexA <> GVL.g_stHMIToolEditorA.LoadedIndex
		AND GVL.g_aToolConfigA[GVL.g_uiHMIToolCheckIndexA].Enable
        AND GVL.g_aToolConfigA[GVL.g_uiHMIToolCheckIndexA].ToolID = GVL.g_stHMIToolEditorA.EditData.ToolID THEN

            GVL.g_xHMIToolDuplicateIDA := TRUE;

        END_IF;

    END_FOR;

    //-------------------------------------------------------------------------
    // Kiểm tra dữ liệu trước khi Save.
    //-------------------------------------------------------------------------
    IF GVL.g_stHMIToolEditorA.LoadedIndex < 1
    OR GVL.g_stHMIToolEditorA.LoadedIndex > GVL.C_MAX_TOOLS THEN

        GVL.g_stHMIToolEditorA.Error := TRUE;
        GVL.g_stHMIToolEditorA.ErrorID := 1110;

    ELSIF GVL.g_stMultiTrackStatusA.Busy THEN

        // Không cho thay cấu hình khi Multi-tool đang chạy.
        GVL.g_stHMIToolEditorA.Error := TRUE;
        GVL.g_stHMIToolEditorA.ErrorID := 1111;

    ELSIF GVL.g_aToolStatusA[GVL.g_stHMIToolEditorA.LoadedIndex].Busy THEN

        // Không cho thay cấu hình khi Tool đang thực hiện lệnh.
        GVL.g_stHMIToolEditorA.Error := TRUE;
        GVL.g_stHMIToolEditorA.ErrorID := 1112;

    ELSIF GVL.g_stHMIToolEditorA.EditData.ToolID = 0 THEN

        GVL.g_stHMIToolEditorA.Error := TRUE;
        GVL.g_stHMIToolEditorA.ErrorID := 1113;

    ELSIF GVL.g_xHMIToolDuplicateIDA THEN

        GVL.g_stHMIToolEditorA.Error := TRUE;
        GVL.g_stHMIToolEditorA.ErrorID := 1114;

    ELSIF GVL.g_stHMIToolEditorA.EditData.ApproachHeight < 0.0 THEN

        GVL.g_stHMIToolEditorA.Error := TRUE;
        GVL.g_stHMIToolEditorA.ErrorID := 1115;

    ELSIF GVL.g_stHMIToolEditorA.EditData.UseUpDown AND GVL.g_stHMIToolEditorA.EditData.UpDownStroke <= 0.0 THEN

        GVL.g_stHMIToolEditorA.Error := TRUE;
        GVL.g_stHMIToolEditorA.ErrorID := 1116;
	ELSIF GVL.g_stHMIToolEditorA.EditData.UseUpDown AND GVL.g_stHMIToolEditorA.EditData.IO.UseSingleUpDownDO
	AND (GVL.g_stHMIToolEditorA.EditData.IO.UpDownDOChannel = 0 OR GVL.g_stHMIToolEditorA.EditData.IO.UpDownDOChannel > GVL.C_MAX_DO) THEN
		GVL.g_stHMIToolEditorA.Error := TRUE;
		GVL.g_stHMIToolEditorA.ErrorID := 1120;
	
	ELSIF GVL.g_stHMIToolEditorA.EditData.UseUpDown AND NOT GVL.g_stHMIToolEditorA.EditData.IO.UseSingleUpDownDO
	AND (GVL.g_stHMIToolEditorA.EditData.IO.DownDOChannel = 0 OR GVL.g_stHMIToolEditorA.EditData.IO.DownDOChannel > GVL.C_MAX_DO) THEN
		GVL.g_stHMIToolEditorA.Error := TRUE;
		GVL.g_stHMIToolEditorA.ErrorID := 1121;
	
	ELSIF GVL.g_stHMIToolEditorA.EditData.UseUpDown AND NOT GVL.g_stHMIToolEditorA.EditData.IO.UseSingleUpDownDO
	AND (GVL.g_stHMIToolEditorA.EditData.IO.UpDOChannel = 0 OR GVL.g_stHMIToolEditorA.EditData.IO.UpDOChannel > GVL.C_MAX_DO) THEN
		GVL.g_stHMIToolEditorA.Error := TRUE;
		GVL.g_stHMIToolEditorA.ErrorID := 1122;
	ELSIF GVL.g_stHMIToolEditorA.EditData.IO.UseSingleGripReleaseDO
	AND (
		//GVL.g_stHMIToolEditorA.EditData.IO.GripReleaseDOChannel = 0 OR 
		GVL.g_stHMIToolEditorA.EditData.IO.GripReleaseDOChannel > GVL.C_MAX_DO
	) THEN
		GVL.g_stHMIToolEditorA.Error := TRUE;
		GVL.g_stHMIToolEditorA.ErrorID := 1123;
	
	ELSIF NOT GVL.g_stHMIToolEditorA.EditData.IO.UseSingleGripReleaseDO
	AND GVL.g_stHMIToolEditorA.EditData.IO.GripDOChannel > GVL.C_MAX_DO THEN
		GVL.g_stHMIToolEditorA.Error := TRUE;
		GVL.g_stHMIToolEditorA.ErrorID := 1124;
	
	ELSIF NOT GVL.g_stHMIToolEditorA.EditData.IO.UseSingleGripReleaseDO
	AND GVL.g_stHMIToolEditorA.EditData.IO.ReleaseDOChannel > GVL.C_MAX_DO THEN
		GVL.g_stHMIToolEditorA.Error := TRUE;
		GVL.g_stHMIToolEditorA.ErrorID := 1125;
    ELSE

        // Ghi dữ liệu từ vùng trung gian về đúng Tool đã Load.
        GVL.g_aToolConfigA[GVL.g_stHMIToolEditorA.LoadedIndex] := GVL.g_stHMIToolEditorA.EditData;

        // Cập nhật bản gốc sau khi Save thành công.
        GVL.g_stHMIToolEditorA.OriginalData := GVL.g_stHMIToolEditorA.EditData;

        GVL.g_stHMIToolEditorA.DataChanged := FALSE;
        GVL.g_stHMIToolEditorA.SaveDone := TRUE;
		GVL.g_stHMITool_Config_Save_All := TRUE;

    END_IF;

END_IF;


//=============================================================================
// 08. CẬP NHẬT TRẠNG THÁI TOOL ĐƯỢC CHỌN
//-----------------------------------------------------------------------------
// HMI đọc một biến cố định thay vì dùng địa chỉ mảng động.
//=============================================================================
IF GVL.g_stHMIToolEditorA.LoadedIndex >= 1
AND GVL.g_stHMIToolEditorA.LoadedIndex <= GVL.C_MAX_TOOLS THEN

    GVL.g_stHMIToolStatusA :=
        GVL.g_aToolStatusA[
            GVL.g_stHMIToolEditorA.LoadedIndex
        ];

END_IF;
END_ACTION

ACTION ACT_HMIToolConfigEditor_B:
// CREATE ACTION under POU_HMI_CONTROL_ROBOT: ACT_HMIToolConfigEditor_B

//=============================================================================
// PROGRAM: PRG_HMIToolConfigEditor_B
//-----------------------------------------------------------------------------
// Quản lý trang HMI cấu hình nhiều Tool cho Robot B.
//
// NGUYÊN TẮC:
// 1. HMI chỉnh EditData, không chỉnh trực tiếp g_aToolConfigB.
// 2. Load sao chép ToolConfig vào EditData.
// 3. Save kiểm tra dữ liệu rồi mới ghi về ToolConfig.
// 4. Cancel khôi phục dữ liệu từ OriginalData.
// 5. Save luôn ghi theo LoadedIndex để tránh ghi nhầm Tool.
//=============================================================================


//=============================================================================
// 01. BẮT CẠNH LỆNH HMI
//=============================================================================
GVL.g_rtHMIToolLoadB(CLK := GVL.g_stHMIToolEditorB.LoadCommand);

GVL.g_rtHMIToolSaveB(CLK := GVL.g_stHMIToolEditorB.SaveCommand);

GVL.g_rtHMIToolCancelB(CLK := GVL.g_stHMIToolEditorB.CancelCommand);


//=============================================================================
// 02. OUTPUT DẠNG XUNG
//-----------------------------------------------------------------------------
// LoadDone và SaveDone chỉ TRUE trong một vòng quét.
//=============================================================================
GVL.g_stHMIToolEditorB.LoadDone := FALSE;
GVL.g_stHMIToolEditorB.SaveDone := FALSE;
GVL.g_stHMIToolEditorB.Busy := FALSE;


//=============================================================================
// 03. KHỞI TẠO INDEX MẶC ĐỊNH
//=============================================================================
IF GVL.g_stHMIToolEditorB.SelectedIndex = 0 THEN
    GVL.g_stHMIToolEditorB.SelectedIndex := 1;
END_IF;


//=============================================================================
// 04. TỰ ĐỘNG LOAD KHI ĐỔI TOOL
//-----------------------------------------------------------------------------
// Chỉ tự động Load khi dữ liệu hiện tại chưa bị chỉnh sửa.
// Nếu DataChanged = TRUE thì giữ dữ liệu hiện tại để tránh mất dữ liệu.
//=============================================================================
IF GVL.g_stHMIToolEditorB.SelectedIndex <> GVL.g_uiHMIToolSelectedIndexOldB THEN

    IF GVL.g_stHMIToolEditorB.DataChanged THEN

        // Không cho đổi Tool khi dữ liệu hiện tại chưa được Save hoặc Cancel.
        GVL.g_stHMIToolEditorB.SelectedIndex := GVL.g_uiHMIToolSelectedIndexOldB;

        GVL.g_stHMIToolEditorB.Error := TRUE;
        GVL.g_stHMIToolEditorB.ErrorID := 1101;

    ELSIF GVL.g_stHMIToolEditorB.SelectedIndex >= 1 AND GVL.g_stHMIToolEditorB.SelectedIndex <= GVL.C_MAX_TOOLS THEN

        // Sao chép cấu hình Tool được chọn vào vùng chỉnh sửa.
        GVL.g_stHMIToolEditorB.EditData := GVL.g_aToolConfigB[GVL.g_stHMIToolEditorB.SelectedIndex];

        // Lưu bản gốc để phục vụ Cancel.
        GVL.g_stHMIToolEditorB.OriginalData := GVL.g_aToolConfigB[GVL.g_stHMIToolEditorB.SelectedIndex];

        GVL.g_stHMIToolEditorB.LoadedIndex := GVL.g_stHMIToolEditorB.SelectedIndex;

        GVL.g_uiHMIToolSelectedIndexOldB := GVL.g_stHMIToolEditorB.SelectedIndex;

        GVL.g_stHMIToolEditorB.DataChanged := FALSE;
        GVL.g_stHMIToolEditorB.Error := FALSE;
        GVL.g_stHMIToolEditorB.ErrorID := 0;
        GVL.g_stHMIToolEditorB.LoadDone := TRUE;

    ELSE

        // Index Tool ngoài phạm vi.
        GVL.g_stHMIToolEditorB.Error := TRUE;
        GVL.g_stHMIToolEditorB.ErrorID := 1102;

    END_IF;

END_IF;


//=============================================================================
// 05. LOAD THỦ CÔNG
//=============================================================================
IF GVL.g_rtHMIToolLoadB.Q THEN

    GVL.g_stHMIToolEditorB.Busy := TRUE;
    GVL.g_stHMIToolEditorB.Error := FALSE;
    GVL.g_stHMIToolEditorB.ErrorID := 0;

    IF GVL.g_stHMIToolEditorB.SelectedIndex >= 1
    AND GVL.g_stHMIToolEditorB.SelectedIndex <= GVL.C_MAX_TOOLS THEN

        GVL.g_stHMIToolEditorB.EditData := GVL.g_aToolConfigB[GVL.g_stHMIToolEditorB.SelectedIndex];

        GVL.g_stHMIToolEditorB.OriginalData := GVL.g_aToolConfigB[GVL.g_stHMIToolEditorB.SelectedIndex];

        GVL.g_stHMIToolEditorB.LoadedIndex := GVL.g_stHMIToolEditorB.SelectedIndex;

        GVL.g_uiHMIToolSelectedIndexOldB := GVL.g_stHMIToolEditorB.SelectedIndex;

        GVL.g_stHMIToolEditorB.DataChanged := FALSE;
        GVL.g_stHMIToolEditorB.LoadDone := TRUE;

    ELSE

        GVL.g_stHMIToolEditorB.Error := TRUE;
        GVL.g_stHMIToolEditorB.ErrorID := 1102;

    END_IF;
	
	GVL.g_stHMIToolEditorB.LoadCommand := FALSE;

END_IF;


// //=============================================================================
// // 06. CANCEL THAY ĐỔI
// //-----------------------------------------------------------------------------
// // Khôi phục EditData về bản dữ liệu đã Load gần nhất.
// //=============================================================================
// IF GVL.g_rtHMIToolCancelB.Q THEN
// 
//     GVL.g_stHMIToolEditorB.Busy := TRUE;
//     GVL.g_stHMIToolEditorB.Error := FALSE;
//     GVL.g_stHMIToolEditorB.ErrorID := 0;
// 
//     IF GVL.g_stHMIToolEditorB.LoadedIndex >= 1
//     AND GVL.g_stHMIToolEditorB.LoadedIndex <= GVL.C_MAX_TOOLS THEN
// 
//         GVL.g_stHMIToolEditorB.EditData := GVL.g_stHMIToolEditorB.OriginalData;
// 
//         GVL.g_stHMIToolEditorB.DataChanged := FALSE;
//         GVL.g_stHMIToolEditorB.LoadDone := TRUE;
// 
//     ELSE
// 
//         GVL.g_stHMIToolEditorB.Error := TRUE;
//         GVL.g_stHMIToolEditorB.ErrorID := 1103;
// 
//     END_IF;
// 
// END_IF;


//=============================================================================
// 07. SAVE CẤU HÌNH TOOL
//=============================================================================
IF GVL.g_rtHMIToolSaveB.Q THEN

    GVL.g_stHMIToolEditorB.Busy := TRUE;
    GVL.g_stHMIToolEditorB.Error := FALSE;
    GVL.g_stHMIToolEditorB.ErrorID := 0;
    GVL.g_xHMIToolDuplicateIDB := FALSE;

    //-------------------------------------------------------------------------
    // Kiểm tra ToolID có trùng với Tool khác hay không.
    //-------------------------------------------------------------------------
    FOR GVL.g_uiHMIToolCheckIndexB := 1 TO GVL.C_MAX_TOOLS DO

        IF GVL.g_uiHMIToolCheckIndexB <> GVL.g_stHMIToolEditorB.LoadedIndex
		AND GVL.g_aToolConfigB[GVL.g_uiHMIToolCheckIndexB].Enable
        AND GVL.g_aToolConfigB[GVL.g_uiHMIToolCheckIndexB].ToolID = GVL.g_stHMIToolEditorB.EditData.ToolID THEN

            GVL.g_xHMIToolDuplicateIDB := TRUE;

        END_IF;

    END_FOR;

    //-------------------------------------------------------------------------
    // Kiểm tra dữ liệu trước khi Save.
    //-------------------------------------------------------------------------
    IF GVL.g_stHMIToolEditorB.LoadedIndex < 1
    OR GVL.g_stHMIToolEditorB.LoadedIndex > GVL.C_MAX_TOOLS THEN

        GVL.g_stHMIToolEditorB.Error := TRUE;
        GVL.g_stHMIToolEditorB.ErrorID := 1110;

    ELSIF GVL.g_stMultiTrackStatusB.Busy THEN

        // Không cho thay cấu hình khi Multi-tool đang chạy.
        GVL.g_stHMIToolEditorB.Error := TRUE;
        GVL.g_stHMIToolEditorB.ErrorID := 1111;

    ELSIF GVL.g_aToolStatusB[GVL.g_stHMIToolEditorB.LoadedIndex].Busy THEN

        // Không cho thay cấu hình khi Tool đang thực hiện lệnh.
        GVL.g_stHMIToolEditorB.Error := TRUE;
        GVL.g_stHMIToolEditorB.ErrorID := 1112;

    ELSIF GVL.g_stHMIToolEditorB.EditData.ToolID = 0 THEN

        GVL.g_stHMIToolEditorB.Error := TRUE;
        GVL.g_stHMIToolEditorB.ErrorID := 1113;

    ELSIF GVL.g_xHMIToolDuplicateIDB THEN

        GVL.g_stHMIToolEditorB.Error := TRUE;
        GVL.g_stHMIToolEditorB.ErrorID := 1114;

    ELSIF GVL.g_stHMIToolEditorB.EditData.ApproachHeight < 0.0 THEN

        GVL.g_stHMIToolEditorB.Error := TRUE;
        GVL.g_stHMIToolEditorB.ErrorID := 1115;

    ELSIF GVL.g_stHMIToolEditorB.EditData.UseUpDown AND GVL.g_stHMIToolEditorB.EditData.UpDownStroke <= 0.0 THEN

        GVL.g_stHMIToolEditorB.Error := TRUE;
        GVL.g_stHMIToolEditorB.ErrorID := 1116;
	ELSIF GVL.g_stHMIToolEditorB.EditData.UseUpDown AND GVL.g_stHMIToolEditorB.EditData.IO.UseSingleUpDownDO
	AND (GVL.g_stHMIToolEditorB.EditData.IO.UpDownDOChannel = 0 OR GVL.g_stHMIToolEditorB.EditData.IO.UpDownDOChannel > GVL.C_MAX_DO) THEN
		GVL.g_stHMIToolEditorB.Error := TRUE;
		GVL.g_stHMIToolEditorB.ErrorID := 1120;
	
	ELSIF GVL.g_stHMIToolEditorB.EditData.UseUpDown AND NOT GVL.g_stHMIToolEditorB.EditData.IO.UseSingleUpDownDO
	AND (GVL.g_stHMIToolEditorB.EditData.IO.DownDOChannel = 0 OR GVL.g_stHMIToolEditorB.EditData.IO.DownDOChannel > GVL.C_MAX_DO) THEN
		GVL.g_stHMIToolEditorB.Error := TRUE;
		GVL.g_stHMIToolEditorB.ErrorID := 1121;
	
	ELSIF GVL.g_stHMIToolEditorB.EditData.UseUpDown AND NOT GVL.g_stHMIToolEditorB.EditData.IO.UseSingleUpDownDO
	AND (GVL.g_stHMIToolEditorB.EditData.IO.UpDOChannel = 0 OR GVL.g_stHMIToolEditorB.EditData.IO.UpDOChannel > GVL.C_MAX_DO) THEN
		GVL.g_stHMIToolEditorB.Error := TRUE;
		GVL.g_stHMIToolEditorB.ErrorID := 1122;
	ELSIF GVL.g_stHMIToolEditorB.EditData.IO.UseSingleGripReleaseDO
	AND (
		//GVL.g_stHMIToolEditorB.EditData.IO.GripReleaseDOChannel = 0 OR 
		GVL.g_stHMIToolEditorB.EditData.IO.GripReleaseDOChannel > GVL.C_MAX_DO
	) THEN
		GVL.g_stHMIToolEditorB.Error := TRUE;
		GVL.g_stHMIToolEditorB.ErrorID := 1123;
	
	ELSIF NOT GVL.g_stHMIToolEditorB.EditData.IO.UseSingleGripReleaseDO
	AND GVL.g_stHMIToolEditorB.EditData.IO.GripDOChannel > GVL.C_MAX_DO THEN
		GVL.g_stHMIToolEditorB.Error := TRUE;
		GVL.g_stHMIToolEditorB.ErrorID := 1124;
	
	ELSIF NOT GVL.g_stHMIToolEditorB.EditData.IO.UseSingleGripReleaseDO
	AND GVL.g_stHMIToolEditorB.EditData.IO.ReleaseDOChannel > GVL.C_MAX_DO THEN
		GVL.g_stHMIToolEditorB.Error := TRUE;
		GVL.g_stHMIToolEditorB.ErrorID := 1125;
    ELSE

        // Ghi dữ liệu từ vùng trung gian về đúng Tool đã Load.
        GVL.g_aToolConfigB[GVL.g_stHMIToolEditorB.LoadedIndex] := GVL.g_stHMIToolEditorB.EditData;

        // Cập nhật bản gốc sau khi Save thành công.
        GVL.g_stHMIToolEditorB.OriginalData := GVL.g_stHMIToolEditorB.EditData;

        GVL.g_stHMIToolEditorB.DataChanged := FALSE;
        GVL.g_stHMIToolEditorB.SaveDone := TRUE;
		GVL.g_xHMIToolConfigSaveAllB := TRUE;

    END_IF;

END_IF;


//=============================================================================
// 08. CẬP NHẬT TRẠNG THÁI TOOL ĐƯỢC CHỌN
//-----------------------------------------------------------------------------
// HMI đọc một biến cố định thay vì dùng địa chỉ mảng động.
//=============================================================================
IF GVL.g_stHMIToolEditorB.LoadedIndex >= 1
AND GVL.g_stHMIToolEditorB.LoadedIndex <= GVL.C_MAX_TOOLS THEN

    GVL.g_stHMIToolStatusB :=
        GVL.g_aToolStatusB[
            GVL.g_stHMIToolEditorB.LoadedIndex
        ];

END_IF;
END_ACTION

ACTION ACT_JOG_LOGIC:
// CONTINUE --- INCHING ----POINT
//  RB_A

TRIG_JOG_CONTINUE_1(CLK:= GVL.RB_A.Jog_continue);
TRIG_JOG_INCHING_1(CLK:= GVL.RB_A.Jog_Inching);
TRIG_JOG_POINT_1(CLK:= GVL.RB_A.Jog_Point);
// 
RS_JOG_CONTINUE_1(
    SET1  := TRIG_JOG_CONTINUE_1.Q  ,
    RESET := TRIG_JOG_INCHING_1.Q OR TRIG_JOG_POINT_1.Q,
    Q1    => GVL.RB_A.Jog_continue
);

RS_JOG_INCHING_1(
    SET1  := TRIG_JOG_INCHING_1.Q,
    RESET := TRIG_JOG_CONTINUE_1.Q OR TRIG_JOG_POINT_1.Q,
    Q1    => GVL.RB_A.Jog_Inching
);
RS_JOG_POINT_1(
    SET1  := TRIG_JOG_POINT_1.Q,
    RESET := TRIG_JOG_CONTINUE_1.Q OR TRIG_JOG_INCHING_1.Q,
    Q1    => GVL.RB_A.Jog_Point
);
// RB_B	
			   
TRIG_JOG_CONTINUE_2(CLK:= GVL.RB_B.Jog_continue );
TRIG_JOG_INCHING_2(CLK:= GVL.RB_B.Jog_Inching);
TRIG_JOG_POINT_2(CLK:= GVL.RB_B.Jog_Point);
// 
RS_JOG_CONTINUE_2(
    SET1  := TRIG_JOG_CONTINUE_2.Q,
    RESET := TRIG_JOG_INCHING_2.Q OR TRIG_JOG_POINT_2.Q,
    Q1    => GVL.RB_B.Jog_continue
);

RS_JOG_INCHING_2(
    SET1  := TRIG_JOG_INCHING_2.Q,
    RESET := TRIG_JOG_CONTINUE_2.Q OR TRIG_JOG_POINT_2.Q,
    Q1    => GVL.RB_B.Jog_Inching
);

RS_JOG_POINT_2(
    SET1  := TRIG_JOG_POINT_2.Q,
    RESET := TRIG_JOG_CONTINUE_2.Q OR TRIG_JOG_INCHING_2.Q,
    Q1    => GVL.RB_B.Jog_Point
);
END_ACTION

ACTION ACT_MANORAUTO:
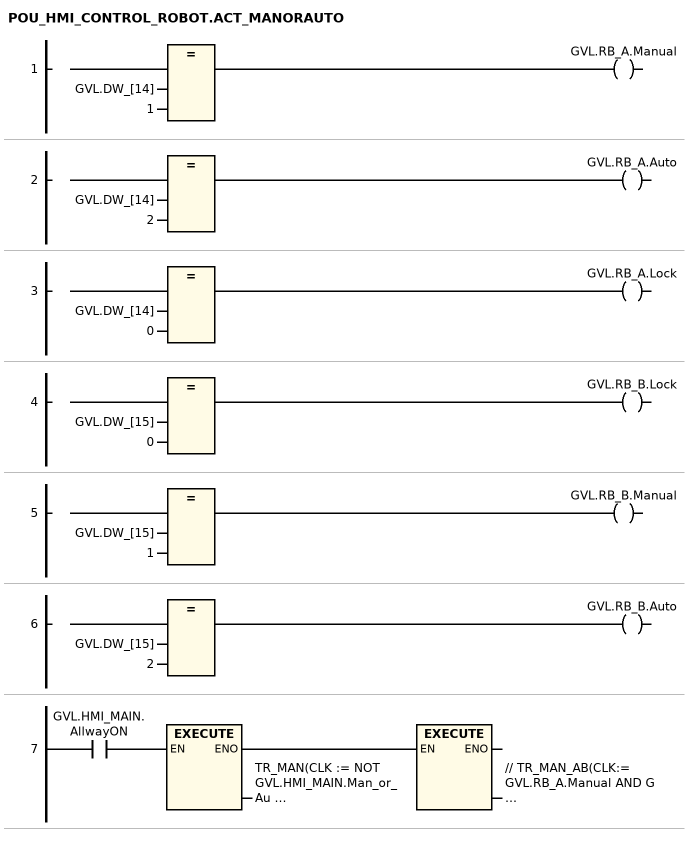
// NETWORK 1
GVL.RB_A.Manual := GVL.DW_[14] = 1;

// NETWORK 2
GVL.RB_A.Auto := GVL.DW_[14] = 2;

// NETWORK 3
GVL.RB_A.Lock := GVL.DW_[14] = 0;

// NETWORK 4
GVL.RB_B.Lock := GVL.DW_[15] = 0;

// NETWORK 5
GVL.RB_B.Manual := GVL.DW_[15] = 1;

// NETWORK 6
GVL.RB_B.Auto := GVL.DW_[15] = 2;

// NETWORK 7
_w1 := GVL.HMI_MAIN.AllwayON;
IF _w1 THEN
    TR_MAN(CLK := NOT GVL.HMI_MAIN.Man_or_Auto);
    TR_AUTO(CLK := GVL.HMI_MAIN.Man_or_Auto);
    IF TR_AUTO.Q THEN
    	GVL.DW_[14] := 2;
    	GVL.DW_[15] := 2;
    END_IF;
    IF TR_MAN.Q THEN
    	GVL.DW_[14] := 1;
    	GVL.DW_[15] := 1;
    END_IF;
END_IF
IF _w1 THEN
    // TR_MAN_AB(CLK:= GVL.RB_A.Manual AND GVL.RB_B.Manual);
    // TR_AUTO_AB(CLK:=  GVL.RB_A.Auto AND GVL.RB_B.Auto);
    // IF TR_AUTO_AB.Q THEN
    // 	GVL.HMI_MAIN.Man_or_Auto := TRUE;
    // END_IF;
    // IF TR_MAN_AB.Q THEN
    // 	GVL.HMI_MAIN.Man_or_Auto := FALSE;
    // END_IF;
END_IF
END_ACTION

ACTION ACT_MENU:
IF D_SELECT_RB <> PrevSelectRB THEN
    CASE D_SELECT_RB OF
        0: //D_PLC_SCREEN := 20;  // ROBOT_A_PANEL
			IF D_HMI_SCREEN = 31 THEN D_PLC_SCREEN := 21; END_IF;
			IF D_HMI_SCREEN = 32 THEN D_PLC_SCREEN := 22; END_IF;		
			IF D_HMI_SCREEN = 33 THEN D_PLC_SCREEN := 23; END_IF;
			IF D_HMI_SCREEN = 34 THEN D_PLC_SCREEN := 24; END_IF;
			IF D_HMI_SCREEN = 35 THEN D_PLC_SCREEN := 25; END_IF;
			IF D_HMI_SCREEN = 36 THEN D_PLC_SCREEN := 26; END_IF;
			IF D_HMI_SCREEN = 30 OR ( D_HMI_SCREEN < 30 OR D_HMI_SCREEN > 36) THEN D_PLC_SCREEN := 20; END_IF;
        1: //D_PLC_SCREEN := 30;  // ROBOT_B_PANEL
			IF D_HMI_SCREEN = 21 THEN D_PLC_SCREEN := 31; END_IF;
			IF D_HMI_SCREEN = 22 THEN D_PLC_SCREEN := 32; END_IF;		
			IF D_HMI_SCREEN = 23 THEN D_PLC_SCREEN := 33; END_IF;
			IF D_HMI_SCREEN = 24 THEN D_PLC_SCREEN := 34; END_IF;
			IF D_HMI_SCREEN = 25 THEN D_PLC_SCREEN := 35; END_IF;
			IF D_HMI_SCREEN = 26 THEN D_PLC_SCREEN := 36; END_IF;
			IF D_HMI_SCREEN = 20 OR ( D_HMI_SCREEN < 20 OR D_HMI_SCREEN > 26) THEN D_PLC_SCREEN := 30; END_IF;		
        2: D_PLC_SCREEN := 100; // R_PANEL
    END_CASE;
END_IF;

PrevSelectRB := D_SELECT_RB;
END_ACTION

ACTION ACT_select_rb:
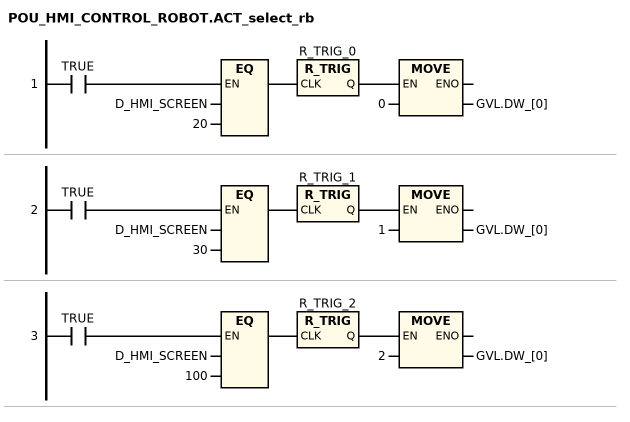
// NETWORK 1
R_TRIG_0(CLK := D_HMI_SCREEN = 20); // R_TRIG
IF R_TRIG_0.Q THEN GVL.DW_[0] := 0; END_IF

// NETWORK 2
R_TRIG_1(CLK := D_HMI_SCREEN = 30); // R_TRIG
IF R_TRIG_1.Q THEN GVL.DW_[0] := 1; END_IF

// NETWORK 3
R_TRIG_2(CLK := D_HMI_SCREEN = 100); // R_TRIG
IF R_TRIG_2.Q THEN GVL.DW_[0] := 2; END_IF
END_ACTION

ACTION ACT_View_Edit_Cmd:
// Lua chon Cac diem can View va Edit 
// CASE GVL.HMI_A_PointViewCmd OF
//     1:
//         GVL.HMI_A_ViewStartPoint := MAX(1, GVL.HMI_A_ViewStartPoint - 1);
// 
//     2:
//         GVL.HMI_A_ViewStartPoint := MIN(491, GVL.HMI_A_ViewStartPoint + 1);
// 
//     3:
//         GVL.HMI_A_ViewStartPoint := MAX(1, GVL.HMI_A_ViewStartPoint - 10);
// 
//     4:
//         GVL.HMI_A_ViewStartPoint := MIN(491, GVL.HMI_A_ViewStartPoint + 10);
// 
//     5:
//         GVL.HMI_A_ViewStartPoint := 1;
// 
//     6:
//         GVL.HMI_A_ViewStartPoint := 491;
// 
// END_CASE;
// 
// GVL.HMI_A_PointViewCmd := 0;

// // Up 1
// IF GVL.HMI_A_ViewCmd_Scroll_Up AND NOT GVL.HMI_A_ViewCmd_Scroll_Up_Old THEN
// 	GVL.HMI_A_ViewStartStep := MAX (1, GVL.HMI_A_ViewStartStep - 1);
// END_IF
// GVL.HMI_A_ViewCmd_Scroll_Up_Old := GVL.HMI_A_ViewCmd_Scroll_Up;
// // Down 1
// IF GVL.HMI_A_ViewCmd_Scroll_Down AND NOT GVL.HMI_A_ViewCmd_Scroll_Down_Old THEN
// 	GVL.HMI_A_ViewStartStep := MAX (1, GVL.HMI_A_ViewStartStep + 1);
// END_IF
// GVL.HMI_A_ViewCmd_Scroll_Down_Old := GVL.HMI_A_ViewCmd_Scroll_Down;
// // Up 10
// IF GVL.HMI_A_ViewCmd_Page_Up AND NOT GVL.HMI_A_ViewCmd_Page_Up_Old THEN
// 	GVL.HMI_A_ViewStartStep := MAX (1, GVL.HMI_A_ViewStartStep - 10);
// END_IF
// GVL.HMI_A_ViewCmd_Page_Up_Old := GVL.HMI_A_ViewCmd_Page_Up;
// // Down 10
// IF GVL.HMI_A_ViewCmd_Page_Down AND NOT GVL.HMI_A_ViewCmd_Page_Down_Old THEN
// 	GVL.HMI_A_ViewStartStep := MAX (1, GVL.HMI_A_ViewStartStep + 10);
// END_IF
// GVL.HMI_A_ViewCmd_Page_Down_Old := GVL.HMI_A_ViewCmd_Page_Down;
// // Up Top
// IF GVL.HMI_A_ViewCmd_Go_Top AND NOT GVL.HMI_A_ViewCmd_Go_Top_Old THEN
// 	GVL.HMI_A_ViewStartStep := 1;
// END_IF
// GVL.HMI_A_ViewCmd_Go_Top_Old := GVL.HMI_A_ViewCmd_Go_Top;
// // Down Bot
// IF GVL.HMI_A_ViewCmd_Go_Bot AND NOT GVL.HMI_A_ViewCmd_Go_Bot_Old THEN
// 	GVL.HMI_A_ViewStartStep := GVL.A_LengthStep - 9;
// END_IF
// GVL.HMI_A_ViewCmd_Go_Bot_Old := GVL.HMI_A_ViewCmd_Go_Bot;

// Up 1
IF GVL.HMI_A_ViewCmd_Scroll_Up THEN
	GVL.HMI_A_ViewStartStep := MAX (1, GVL.HMI_A_ViewStartStep - 1);
END_IF
GVL.HMI_A_ViewCmd_Scroll_Up := FALSE;
// Down 1
IF GVL.HMI_A_ViewCmd_Scroll_Down THEN
	GVL.HMI_A_ViewStartStep := MAX (1, GVL.HMI_A_ViewStartStep + 1);
END_IF
GVL.HMI_A_ViewCmd_Scroll_Down := FALSE;
// Up 10
IF GVL.HMI_A_ViewCmd_Page_Up THEN
	GVL.HMI_A_ViewStartStep := MAX (1, GVL.HMI_A_ViewStartStep - 10);
	GVL.HMI_A_RowSelectedCmd := 0;
END_IF
GVL.HMI_A_ViewCmd_Page_Up := FALSE;
// Down 10
IF GVL.HMI_A_ViewCmd_Page_Down THEN
	GVL.HMI_A_ViewStartStep := MAX (1, GVL.HMI_A_ViewStartStep + 10);
	GVL.HMI_A_RowSelectedCmd := 0;
END_IF
GVL.HMI_A_ViewCmd_Page_Down := FALSE;
// Up Top
IF GVL.HMI_A_ViewCmd_Go_Top THEN
	GVL.HMI_A_ViewStartStep := 1;
	GVL.HMI_A_RowSelectedCmd := 0;
END_IF
GVL.HMI_A_ViewCmd_Go_Top := FALSE;
// Down Bot
IF GVL.HMI_A_ViewCmd_Go_Bot THEN
	GVL.HMI_A_ViewStartStep := MAX(1, GVL.A_LengthStep - 9);
	GVL.HMI_A_RowSelectedCmd := 0;
END_IF
GVL.HMI_A_ViewCmd_Go_Bot := FALSE;


// Refresh 10 dòng
FOR i := 1 TO 10 DO
    idx := GVL.HMI_A_ViewStartStep + i - 1;

    GVL.HMI_A_ViewStepNo[i]   := idx;
    GVL.HMI_A_ViewGroupCmd[i] := GVL_1.Step_Cr_A[idx].GroupCmd;
    GVL.HMI_A_ViewCmd[i]      := TO_INT(GVL_1.Step_Cr_A[idx].Cmd);

    GVL.HMI_A_ViewP1[i] := GVL_1.Step_Cr_A[idx].P1;
    GVL.HMI_A_ViewP2[i] := GVL_1.Step_Cr_A[idx].P2;
    GVL.HMI_A_ViewP3[i] := GVL_1.Step_Cr_A[idx].P3;
    GVL.HMI_A_ViewP4[i] := GVL_1.Step_Cr_A[idx].P4;
    GVL.HMI_A_ViewP5[i] := GVL_1.Step_Cr_A[idx].P5;
    GVL.HMI_A_ViewP6[i] := GVL_1.Step_Cr_A[idx].P6;

    GVL.HMI_A_ViewNote[i] := GVL_1.Step_Cr_A[idx].Note;
END_FOR;

// Refresh command hien thi tren HMI
FOR i := 1 TO 10 DO
    idx := GVL.HMI_A_ViewStartStep + i - 1;

    GVL.HMI_A_ViewStepNo[i]   := idx;
    GVL.HMI_A_ViewCmd[i]      := TO_INT(GVL_1.Step_Cr_A[idx].Cmd);
    GVL.HMI_A_ViewP1[i]       := GVL_1.Step_Cr_A[idx].P1;
	GVL.HMI_A_ViewP2[i]       := GVL_1.Step_Cr_A[idx].P2;
	GVL.HMI_A_ViewP3[i]       := GVL_1.Step_Cr_A[idx].P3;
	GVL.HMI_A_ViewP4[i]       := GVL_1.Step_Cr_A[idx].P4;
	GVL.HMI_A_ViewP5[i]       := GVL_1.Step_Cr_A[idx].P5;
	GVL.HMI_A_ViewNote[i]     := GVL_1.Step_Cr_A[idx].Note;
END_FOR

// Tinh diem lua chon thuc te tren PLC tu HMI
//GVL.HMI_A_Poi := HMI_PointStartIndex + HMI_PointSelectedRow - 1;

// Xu ly chon dong
FOR i := 1 TO 10 DO
	IF NOT GVL.A_RunEnable THEN
		IF (GVL.HMI_A_RowSelectedCmd = i) THEN
			GVL.HMI_A_RowSelect[i] := TRUE;
			GVL.HMI_A_SelectedStepNo := i + GVL.HMI_A_ViewStartStep - 1;
			GVL.HMI_A_EditStepNo   := GVL.HMI_A_SelectedStepNo;
		ELSE
			GVL.HMI_A_RowSelect[i] := FALSE;
		END_IF;
	ELSE
		IF (GVL.A_RunStep = i) THEN
			GVL.HMI_A_RowSelect[i] := TRUE;
		ELSE
			GVL.HMI_A_RowSelect[i] := FALSE;
		END_IF
	END_IF
END_FOR;

// Tao bien de chon windown edit command

FOR i := 0 TO 10 DO
	IF GVL.HMI_A_EditGroupCmd = i THEN
		GVL.HMI_A_Edit_Trigger_Windown_Cmd[i] := TRUE;
	ELSE
		GVL.HMI_A_Edit_Trigger_Windown_Cmd[i] := FALSE;
	END_IF
END_FOR;

// Edit Point
CASE GVL.HMI_A_EditCmdReq OF
	// Load Command to Edit
	20:
		//GVL.HMI_A_EditStepNo   := GVL.HMI_A_SelectedStepNo;
		GVL.HMI_A_EditGroupCmd := GVL_1.Step_Cr_A[GVL.HMI_A_SelectedStepNo].GroupCmd;
		GVL.HMI_A_EditCmd      := GVL_1.Step_Cr_A[GVL.HMI_A_SelectedStepNo].Cmd;
		GVL.HMI_A_EditP1       := GVL_1.Step_Cr_A[GVL.HMI_A_SelectedStepNo].P1;
		GVL.HMI_A_EditP2       := GVL_1.Step_Cr_A[GVL.HMI_A_SelectedStepNo].P2;
		GVL.HMI_A_EditP3       := GVL_1.Step_Cr_A[GVL.HMI_A_SelectedStepNo].P3;
		GVL.HMI_A_EditP4       := GVL_1.Step_Cr_A[GVL.HMI_A_SelectedStepNo].P4;
		GVL.HMI_A_EditP5       := GVL_1.Step_Cr_A[GVL.HMI_A_SelectedStepNo].P5;
		GVL.HMI_A_EditNote     := GVL_1.Step_Cr_A[GVL.HMI_A_SelectedStepNo].Note;
	
		GVL.HMI_A_EditCmdReq := 0;

	// Save Command Data Edit to PLC
	24:
		//GVL.HMI_A_SelectedStepNo := GVL.HMI_A_EditStepNo;
		GVL_1.Step_Cr_A[GVL.HMI_A_EditStepNo].GroupCmd := GVL.HMI_A_EditGroupCmd;
		GVL_1.Step_Cr_A[GVL.HMI_A_EditStepNo].Cmd := GVL.HMI_A_EditCmd;
		GVL_1.Step_Cr_A[GVL.HMI_A_EditStepNo].P1 := GVL.HMI_A_EditP1;
		GVL_1.Step_Cr_A[GVL.HMI_A_EditStepNo].P2 := GVL.HMI_A_EditP2;
		GVL_1.Step_Cr_A[GVL.HMI_A_EditStepNo].P3 := GVL.HMI_A_EditP3;
		GVL_1.Step_Cr_A[GVL.HMI_A_EditStepNo].P4 := GVL.HMI_A_EditP4;
		GVL_1.Step_Cr_A[GVL.HMI_A_EditStepNo].P5 := GVL.HMI_A_EditP5;
		GVL_1.Step_Cr_A[GVL.HMI_A_EditStepNo].Note := GVL.HMI_A_EditNote;
		IF (GVL.HMI_A_EditStepNo > GVL.A_LengthStep) THEN
			GVL.A_LengthStep := GVL.HMI_A_EditStepNo;
		END_IF
		GVL.HMI_A_RowSelectedCmd := 0;
		GVL.HMI_A_EditCmdReq := 0;


	// Add Command Data Edit to PLC
	21:
		//GVL.HMI_A_SelectedStepNo := GVL.HMI_A_EditStepNo ;
		GVL_1.Step_Cr_A[GVL.HMI_A_EditStepNo].GroupCmd := GVL.HMI_A_EditGroupCmd;
		GVL_1.Step_Cr_A[GVL.HMI_A_EditStepNo].Cmd := GVL.HMI_A_EditCmd;
		GVL_1.Step_Cr_A[GVL.HMI_A_EditStepNo].P1 := GVL.HMI_A_EditP1;
		GVL_1.Step_Cr_A[GVL.HMI_A_EditStepNo].P2 := GVL.HMI_A_EditP2;
		GVL_1.Step_Cr_A[GVL.HMI_A_EditStepNo].P3 := GVL.HMI_A_EditP3;
		GVL_1.Step_Cr_A[GVL.HMI_A_EditStepNo].P4 := GVL.HMI_A_EditP4;
		GVL_1.Step_Cr_A[GVL.HMI_A_EditStepNo].P5 := GVL.HMI_A_EditP5;
		GVL_1.Step_Cr_A[GVL.HMI_A_EditStepNo].Note := GVL.HMI_A_EditNote;
		GVL.A_LengthStep := GVL.A_LengthStep + 1;
		GVL.HMI_A_RowSelectedCmd := 0;
		GVL.HMI_A_EditCmdReq := 0;

	// Insert Command Data To Step Table after line selected
	22:
		//GVL.HMI_A_SelectedStepNo := GVL.HMI_A_EditStepNo;
		FOR i := GVL.A_LengthStep TO (GVL.HMI_A_EditStepNo + 1) BY -1 DO
			GVL_1.Step_Cr_A[i+1] := GVL_1.Step_Cr_A[i];
		END_FOR
		GVL_1.Step_Cr_A[GVL.HMI_A_EditStepNo + 1].GroupCmd := 0;
		GVL_1.Step_Cr_A[GVL.HMI_A_EditStepNo + 1].Cmd := 0;
		GVL_1.Step_Cr_A[GVL.HMI_A_EditStepNo + 1].P1 := 0;
		GVL_1.Step_Cr_A[GVL.HMI_A_EditStepNo + 1].P2 := 0;
		GVL_1.Step_Cr_A[GVL.HMI_A_EditStepNo + 1].P3 := 0;
		GVL_1.Step_Cr_A[GVL.HMI_A_EditStepNo + 1].P4 := 0;
		GVL_1.Step_Cr_A[GVL.HMI_A_EditStepNo + 1].P5 := 0;
		GVL_1.Step_Cr_A[GVL.HMI_A_EditStepNo + 1].Note := '';
		GVL.A_LengthStep := GVL.A_LengthStep + 1;
		GVL.HMI_A_EditCmdReq := 0;

// 	// Delete Command Data From Step Table
// 	23:
// 		//GVL.HMI_A_SelectedStepNo := GVL.HMI_A_EditStepNo;
// 		FOR i := (GVL.HMI_A_EditStepNo) TO (GVL.A_LengthStep -1) BY 1 DO
// 			GVL_1.Step_Cr_A[i] := GVL_1.Step_Cr_A[i+1];
// 		END_FOR
// 		GVL_1.Step_Cr_A[GVL.A_LengthStep].GroupCmd := 0;
// 		GVL_1.Step_Cr_A[GVL.A_LengthStep].Cmd := 0;
// 		GVL_1.Step_Cr_A[GVL.A_LengthStep].P1 := 0;
// 		GVL_1.Step_Cr_A[GVL.A_LengthStep].P2 := 0;
// 		GVL_1.Step_Cr_A[GVL.A_LengthStep].P3 := 0;
// 		GVL_1.Step_Cr_A[GVL.A_LengthStep].P4 := 0;
// 		GVL_1.Step_Cr_A[GVL.A_LengthStep].P5 := 0;
// 		GVL_1.Step_Cr_A[GVL.A_LengthStep].Note := '';
// 		GVL.HMI_A_EditCmdReq := 0;
// 		GVL.A_LengthStep := GVL.A_LengthStep - 1;

	//============================================================
	// COPY SINGLE STEP
	// HMI_A_EditCmdReq = 25
	//============================================================
	25:
	
		IF (GVL.HMI_A_SelectedStepNo >= 1)
		   AND (GVL.HMI_A_SelectedStepNo <= GVL.A_LengthStep)
		THEN
	
			GVL.A_StepClipboard :=
				GVL_1.Step_Cr_A[GVL.HMI_A_SelectedStepNo];
	
			GVL.A_StepClipboardValid := TRUE;
	
		END_IF;
	
		GVL.HMI_A_EditCmdReq := 0;
		
	//============================================================
	// PASTE SINGLE STEP
	// Ghi đè vào step đang chọn
	//============================================================
	26:
	
		IF GVL.A_StepClipboardValid	
		   AND (GVL.HMI_A_SelectedStepNo >= 1)
		THEN
	
			GVL_1.Step_Cr_A[GVL.HMI_A_SelectedStepNo] :=
				GVL.A_StepClipboard;
	
			//----------------------------------------------------
			// Nếu paste ra ngoài LengthStep hiện tại
			//----------------------------------------------------
			IF GVL.HMI_A_SelectedStepNo > GVL.A_LengthStep THEN
				GVL.A_LengthStep := GVL.HMI_A_SelectedStepNo;
			END_IF;
	
		END_IF;
	
		GVL.HMI_A_RowSelectedCmd := 0;
		GVL.HMI_A_EditCmdReq := 0;
		
	//============================================================
	// COPY STEP BLOCK
	// HMI_A_EditCmdReq = 28
	//
	// Copy từ HMI_A_CopyStartStep đến HMI_A_CopyEndStep
	//============================================================
	28:
	
		//--------------------------------------------------------
		// Kiểm tra range hợp lệ
		//--------------------------------------------------------
		IF (GVL.HMI_A_CopyStartStep >= 1)
		   AND
		   (GVL.HMI_A_CopyEndStep >= GVL.HMI_A_CopyStartStep)
		   AND
		   (GVL.HMI_A_CopyEndStep <= GVL.A_LengthStep)
		THEN
	
			//----------------------------------------------------
			// Tính số step cần copy
			//----------------------------------------------------
			GVL.AB_StepCopyCount := GVL.HMI_A_CopyEndStep - GVL.HMI_A_CopyStartStep + 1;
	
			//----------------------------------------------------
			// Giới hạn clipboard tối đa 1000 step
			//----------------------------------------------------
			IF GVL.AB_StepCopyCount <= 1000 THEN
	
				FOR i := 1 TO GVL.AB_StepCopyCount DO
	
					GVL.AB_StepBlockClipboard[i] := GVL_1.Step_Cr_A[GVL.HMI_A_CopyStartStep + i - 1];
	
				END_FOR;
	
				//------------------------------------------------
				// Lưu range nguồn để debug / HMI
				//------------------------------------------------
				GVL.A_StepCopyStart := GVL.HMI_A_CopyStartStep;
	
				GVL.A_StepCopyEnd := GVL.HMI_A_CopyEndStep;
	
				GVL.AB_StepBlockClipboardValid := TRUE;
	
			ELSE
	
				//------------------------------------------------
				// Có thể set alarm:
				// block copy quá 100 step
				//------------------------------------------------
				GVL.AB_StepBlockClipboardValid := FALSE;
	
			END_IF;
	
		END_IF;
	
		GVL.HMI_A_EditCmdReq := 0;
		
		//============================================================
	// PASTE STEP BLOCK - INSERT MODE
	// HMI_A_EditCmdReq = 29
	//
	// Ví dụ:
	// clipboard = 5 step
	// Paste tại Step 20
	//
	// Step 20 cũ → 25
	// Step 21 cũ → 26
	// ...
	//
	// Clipboard → Step 20..24
	//============================================================
	29:
	
		IF GVL.AB_StepBlockClipboardValid
		   AND (GVL.AB_StepCopyCount > 0)
		   AND (GVL.HMI_A_SelectedStepNo >= 1)
		THEN
	
			//----------------------------------------------------
			// Kiểm tra không vượt kích thước Step_Cr_A
			//
			// Ví dụ Step_Cr_A[1..500]
			//----------------------------------------------------
			IF (GVL.A_LengthStep + GVL.AB_StepCopyCount) <= 500 THEN
	
				//------------------------------------------------
				// Dịch các step cũ xuống dưới.
				//
				// PHẢI chạy từ dưới lên để không ghi đè dữ liệu.
				//------------------------------------------------
				FOR i := GVL.A_LengthStep TO GVL.HMI_A_SelectedStepNo BY -1 DO
	
					GVL_1.Step_Cr_A[i + GVL.AB_StepCopyCount] := GVL_1.Step_Cr_A[i];
	
				END_FOR;
	
	
				//------------------------------------------------
				// Paste clipboard
				//------------------------------------------------
				FOR i := 1 TO GVL.AB_StepCopyCount DO
	
					GVL_1.Step_Cr_A[GVL.HMI_A_SelectedStepNo + i - 1] := GVL.AB_StepBlockClipboard[i];
	
				END_FOR;
	
	
				//------------------------------------------------
				// Cập nhật tổng số step
				//------------------------------------------------
				GVL.A_LengthStep := GVL.A_LengthStep + GVL.AB_StepCopyCount;
	
	
				//------------------------------------------------
				// Reset select row
				//------------------------------------------------
				GVL.HMI_A_RowSelectedCmd := 0;
	
			END_IF;
	
		END_IF;
	
		GVL.HMI_A_EditCmdReq := 0;
			
END_CASE;

// Delete Command Data From Step Table
Delete_one_Step(IN := GVL.HMI_A_EditCmdReq_Arr[8], PT := T#10MS);
IF Delete_one_Step.Q THEN
	//GVL.HMI_A_SelectedStepNo := GVL.HMI_A_EditStepNo;
	FOR i := (GVL.HMI_A_EditStepNo) TO (GVL.A_LengthStep -1) BY 1 DO
		GVL_1.Step_Cr_A[i] := GVL_1.Step_Cr_A[i+1];
	END_FOR
	GVL_1.Step_Cr_A[GVL.A_LengthStep].GroupCmd := 0;
	GVL_1.Step_Cr_A[GVL.A_LengthStep].Cmd := 0;
	GVL_1.Step_Cr_A[GVL.A_LengthStep].P1 := 0;
	GVL_1.Step_Cr_A[GVL.A_LengthStep].P2 := 0;
	GVL_1.Step_Cr_A[GVL.A_LengthStep].P3 := 0;
	GVL_1.Step_Cr_A[GVL.A_LengthStep].P4 := 0;
	GVL_1.Step_Cr_A[GVL.A_LengthStep].P5 := 0;
	GVL_1.Step_Cr_A[GVL.A_LengthStep].Note := '';
	GVL.HMI_A_EditCmdReq_Arr[8] := FALSE;
	GVL.A_LengthStep := GVL.A_LengthStep - 1;
END_IF

// Delete ALL Command Data From Step Table
Delete_all_Step(IN := GVL.HMI_A_EditCmdReq_Arr[9], PT := T#2S);
IF Delete_all_Step.Q THEN
	//GVL.HMI_A_SelectedStepNo := GVL.HMI_A_EditStepNo;
	FOR i := 0 TO (GVL.A_LengthStep) BY 1 DO
		GVL_1.Step_Cr_A[i].GroupCmd := 0;
		GVL_1.Step_Cr_A[i].Cmd := 0;
		GVL_1.Step_Cr_A[i].P1 := 0;
		GVL_1.Step_Cr_A[i].P2 := 0;
		GVL_1.Step_Cr_A[i].P3 := 0;
		GVL_1.Step_Cr_A[i].P4 := 0;
		GVL_1.Step_Cr_A[i].P5 := 0;
		GVL_1.Step_Cr_A[i].Note := '';
	END_FOR
	
	GVL.HMI_A_EditCmdReq_Arr[8] := FALSE;
	GVL.A_LengthStep := GVL.A_LengthStep - 1;
END_IF


// Enable bit chon nhom lenh
FOR i := 0 TO 10 DO
	IF (GVL.HMI_A_EditGroupCmd >= 0) AND (i = GVL.HMI_A_EditGroupCmd) THEN 
    	GVL.HMI_A_EditSelgroupCmd[i] := TRUE;
	ELSE
		GVL.HMI_A_EditSelgroupCmd[i] := FALSE;
	END_IF
END_FOR;
END_ACTION

ACTION ACT_View_Edit_Cmd_B:
// ============================================================
// CREATE ACTION: ACT_View_Edit_Cmd_B
// Parent POU: POU_HMI_CONTROL_ROBOT
// Source mirrored from: ACT_View_Edit_Cmd
// ============================================================

// Lua chon Cac diem can View va Edit 
// CASE GVL.HMI_B_PointViewCmd OF
//     1:
//         GVL.HMI_B_ViewStartPoint := MAX(1, GVL.HMI_B_ViewStartPoint - 1);
// 
//     2:
//         GVL.HMI_B_ViewStartPoint := MIN(491, GVL.HMI_B_ViewStartPoint + 1);
// 
//     3:
//         GVL.HMI_B_ViewStartPoint := MAX(1, GVL.HMI_B_ViewStartPoint - 10);
// 
//     4:
//         GVL.HMI_B_ViewStartPoint := MIN(491, GVL.HMI_B_ViewStartPoint + 10);
// 
//     5:
//         GVL.HMI_B_ViewStartPoint := 1;
// 
//     6:
//         GVL.HMI_B_ViewStartPoint := 491;
// 
// END_CASE;
// 
// GVL.HMI_B_PointViewCmd := 0;

// // Up 1
// IF GVL.HMI_B_ViewCmd_Scroll_Up AND NOT GVL.HMI_B_ViewCmd_Scroll_Up_Old THEN
// 	GVL.HMI_B_ViewStartStep := MAX (1, GVL.HMI_B_ViewStartStep - 1);
// END_IF
// GVL.HMI_B_ViewCmd_Scroll_Up_Old := GVL.HMI_B_ViewCmd_Scroll_Up;
// // Down 1
// IF GVL.HMI_B_ViewCmd_Scroll_Down AND NOT GVL.HMI_B_ViewCmd_Scroll_Down_Old THEN
// 	GVL.HMI_B_ViewStartStep := MAX (1, GVL.HMI_B_ViewStartStep + 1);
// END_IF
// GVL.HMI_B_ViewCmd_Scroll_Down_Old := GVL.HMI_B_ViewCmd_Scroll_Down;
// // Up 10
// IF GVL.HMI_B_ViewCmd_Page_Up AND NOT GVL.HMI_B_ViewCmd_Page_Up_Old THEN
// 	GVL.HMI_B_ViewStartStep := MAX (1, GVL.HMI_B_ViewStartStep - 10);
// END_IF
// GVL.HMI_B_ViewCmd_Page_Up_Old := GVL.HMI_B_ViewCmd_Page_Up;
// // Down 10
// IF GVL.HMI_B_ViewCmd_Page_Down AND NOT GVL.HMI_B_ViewCmd_Page_Down_Old THEN
// 	GVL.HMI_B_ViewStartStep := MAX (1, GVL.HMI_B_ViewStartStep + 10);
// END_IF
// GVL.HMI_B_ViewCmd_Page_Down_Old := GVL.HMI_B_ViewCmd_Page_Down;
// // Up Top
// IF GVL.HMI_B_ViewCmd_Go_Top AND NOT GVL.HMI_B_ViewCmd_Go_Top_Old THEN
// 	GVL.HMI_B_ViewStartStep := 1;
// END_IF
// GVL.HMI_B_ViewCmd_Go_Top_Old := GVL.HMI_B_ViewCmd_Go_Top;
// // Down Bot
// IF GVL.HMI_B_ViewCmd_Go_Bot AND NOT GVL.HMI_B_ViewCmd_Go_Bot_Old THEN
// 	GVL.HMI_B_ViewStartStep := GVL.B_LengthStep - 9;
// END_IF
// GVL.HMI_B_ViewCmd_Go_Bot_Old := GVL.HMI_B_ViewCmd_Go_Bot;

// Up 1
IF GVL.HMI_B_ViewCmd_Scroll_Up THEN
	GVL.HMI_B_ViewStartStep := MAX (1, GVL.HMI_B_ViewStartStep - 1);
END_IF
GVL.HMI_B_ViewCmd_Scroll_Up := FALSE;
// Down 1
IF GVL.HMI_B_ViewCmd_Scroll_Down THEN
	GVL.HMI_B_ViewStartStep := MAX (1, GVL.HMI_B_ViewStartStep + 1);
END_IF
GVL.HMI_B_ViewCmd_Scroll_Down := FALSE;
// Up 10
IF GVL.HMI_B_ViewCmd_Page_Up THEN
	GVL.HMI_B_ViewStartStep := MAX (1, GVL.HMI_B_ViewStartStep - 10);
	GVL.HMI_B_RowSelectedCmd := 0;
END_IF
GVL.HMI_B_ViewCmd_Page_Up := FALSE;
// Down 10
IF GVL.HMI_B_ViewCmd_Page_Down THEN
	GVL.HMI_B_ViewStartStep := MAX (1, GVL.HMI_B_ViewStartStep + 10);
	GVL.HMI_B_RowSelectedCmd := 0;
END_IF
GVL.HMI_B_ViewCmd_Page_Down := FALSE;
// Up Top
IF GVL.HMI_B_ViewCmd_Go_Top THEN
	GVL.HMI_B_ViewStartStep := 1;
	GVL.HMI_B_RowSelectedCmd := 0;
END_IF
GVL.HMI_B_ViewCmd_Go_Top := FALSE;
// Down Bot
IF GVL.HMI_B_ViewCmd_Go_Bot THEN
	GVL.HMI_B_ViewStartStep := MAX(1, GVL.B_LengthStep - 9);
	GVL.HMI_B_RowSelectedCmd := 0;
END_IF
GVL.HMI_B_ViewCmd_Go_Bot := FALSE;


// Refresh 10 dòng
FOR i := 1 TO 10 DO
    idx := GVL.HMI_B_ViewStartStep + i - 1;

    GVL.HMI_B_ViewStepNo[i]   := idx;
    GVL.HMI_B_ViewGroupCmd[i] := GVL_1.Step_Cr_B[idx].GroupCmd;
    GVL.HMI_B_ViewCmd[i]      := TO_INT(GVL_1.Step_Cr_B[idx].Cmd);

    GVL.HMI_B_ViewP1[i] := GVL_1.Step_Cr_B[idx].P1;
    GVL.HMI_B_ViewP2[i] := GVL_1.Step_Cr_B[idx].P2;
    GVL.HMI_B_ViewP3[i] := GVL_1.Step_Cr_B[idx].P3;
    GVL.HMI_B_ViewP4[i] := GVL_1.Step_Cr_B[idx].P4;
    GVL.HMI_B_ViewP5[i] := GVL_1.Step_Cr_B[idx].P5;
    GVL.HMI_B_ViewP6[i] := GVL_1.Step_Cr_B[idx].P6;

    GVL.HMI_B_ViewNote[i] := GVL_1.Step_Cr_B[idx].Note;
END_FOR;

// Refresh command hien thi tren HMI
FOR i := 1 TO 10 DO
    idx := GVL.HMI_B_ViewStartStep + i - 1;

    GVL.HMI_B_ViewStepNo[i]   := idx;
    GVL.HMI_B_ViewCmd[i]      := TO_INT(GVL_1.Step_Cr_B[idx].Cmd);
    GVL.HMI_B_ViewP1[i]       := GVL_1.Step_Cr_B[idx].P1;
	GVL.HMI_B_ViewP2[i]       := GVL_1.Step_Cr_B[idx].P2;
	GVL.HMI_B_ViewP3[i]       := GVL_1.Step_Cr_B[idx].P3;
	GVL.HMI_B_ViewP4[i]       := GVL_1.Step_Cr_B[idx].P4;
	GVL.HMI_B_ViewP5[i]       := GVL_1.Step_Cr_B[idx].P5;
	GVL.HMI_B_ViewNote[i]     := GVL_1.Step_Cr_B[idx].Note;
END_FOR

// Tinh diem lua chon thuc te tren PLC tu HMI
//GVL.HMI_B_Poi := HMI_PointStartIndex + HMI_PointSelectedRow - 1;

// Xu ly chon dong
FOR i := 1 TO 10 DO
	IF NOT GVL.B_RunEnable THEN
		IF (GVL.HMI_B_RowSelectedCmd = i) THEN
			GVL.HMI_B_RowSelect[i] := TRUE;
			GVL.HMI_B_SelectedStepNo := i + GVL.HMI_B_ViewStartStep - 1;
			GVL.HMI_B_EditStepNo   := GVL.HMI_B_SelectedStepNo;
		ELSE
			GVL.HMI_B_RowSelect[i] := FALSE;
		END_IF;
	ELSE
		IF (GVL.B_RunStep = i) THEN
			GVL.HMI_B_RowSelect[i] := TRUE;
		ELSE
			GVL.HMI_B_RowSelect[i] := FALSE;
		END_IF
	END_IF
END_FOR;

// Tao bien de chon windown edit command

FOR i := 0 TO 10 DO
	IF GVL.HMI_B_EditGroupCmd = i THEN
		GVL.HMI_B_Edit_Trigger_Windown_Cmd[i] := TRUE;
	ELSE
		GVL.HMI_B_Edit_Trigger_Windown_Cmd[i] := FALSE;
	END_IF
END_FOR;

// Edit Point
CASE GVL.HMI_B_EditCmdReq OF
	// Load Command to Edit
	20:
		//GVL.HMI_B_EditStepNo   := GVL.HMI_B_SelectedStepNo;
		GVL.HMI_B_EditGroupCmd := GVL_1.Step_Cr_B[GVL.HMI_B_SelectedStepNo].GroupCmd;
		GVL.HMI_B_EditCmd      := GVL_1.Step_Cr_B[GVL.HMI_B_SelectedStepNo].Cmd;
		GVL.HMI_B_EditP1       := GVL_1.Step_Cr_B[GVL.HMI_B_SelectedStepNo].P1;
		GVL.HMI_B_EditP2       := GVL_1.Step_Cr_B[GVL.HMI_B_SelectedStepNo].P2;
		GVL.HMI_B_EditP3       := GVL_1.Step_Cr_B[GVL.HMI_B_SelectedStepNo].P3;
		GVL.HMI_B_EditP4       := GVL_1.Step_Cr_B[GVL.HMI_B_SelectedStepNo].P4;
		GVL.HMI_B_EditP5       := GVL_1.Step_Cr_B[GVL.HMI_B_SelectedStepNo].P5;
		GVL.HMI_B_EditNote     := GVL_1.Step_Cr_B[GVL.HMI_B_SelectedStepNo].Note;
	
		GVL.HMI_B_EditCmdReq := 0;

	// Save Command Data Edit to PLC
	24:
		//GVL.HMI_B_SelectedStepNo := GVL.HMI_B_EditStepNo;
		GVL_1.Step_Cr_B[GVL.HMI_B_EditStepNo].GroupCmd := GVL.HMI_B_EditGroupCmd;
		GVL_1.Step_Cr_B[GVL.HMI_B_EditStepNo].Cmd := GVL.HMI_B_EditCmd;
		GVL_1.Step_Cr_B[GVL.HMI_B_EditStepNo].P1 := GVL.HMI_B_EditP1;
		GVL_1.Step_Cr_B[GVL.HMI_B_EditStepNo].P2 := GVL.HMI_B_EditP2;
		GVL_1.Step_Cr_B[GVL.HMI_B_EditStepNo].P3 := GVL.HMI_B_EditP3;
		GVL_1.Step_Cr_B[GVL.HMI_B_EditStepNo].P4 := GVL.HMI_B_EditP4;
		GVL_1.Step_Cr_B[GVL.HMI_B_EditStepNo].P5 := GVL.HMI_B_EditP5;
		GVL_1.Step_Cr_B[GVL.HMI_B_EditStepNo].Note := GVL.HMI_B_EditNote;
		IF (GVL.HMI_B_EditStepNo > GVL.B_LengthStep) THEN
			GVL.B_LengthStep := GVL.HMI_B_EditStepNo;
		END_IF
		GVL.HMI_B_RowSelectedCmd := 0;
		GVL.HMI_B_EditCmdReq := 0;


	// Add Command Data Edit to PLC
	21:
		//GVL.HMI_B_SelectedStepNo := GVL.HMI_B_EditStepNo ;
		GVL_1.Step_Cr_B[GVL.HMI_B_EditStepNo].GroupCmd := GVL.HMI_B_EditGroupCmd;
		GVL_1.Step_Cr_B[GVL.HMI_B_EditStepNo].Cmd := GVL.HMI_B_EditCmd;
		GVL_1.Step_Cr_B[GVL.HMI_B_EditStepNo].P1 := GVL.HMI_B_EditP1;
		GVL_1.Step_Cr_B[GVL.HMI_B_EditStepNo].P2 := GVL.HMI_B_EditP2;
		GVL_1.Step_Cr_B[GVL.HMI_B_EditStepNo].P3 := GVL.HMI_B_EditP3;
		GVL_1.Step_Cr_B[GVL.HMI_B_EditStepNo].P4 := GVL.HMI_B_EditP4;
		GVL_1.Step_Cr_B[GVL.HMI_B_EditStepNo].P5 := GVL.HMI_B_EditP5;
		GVL_1.Step_Cr_B[GVL.HMI_B_EditStepNo].Note := GVL.HMI_B_EditNote;
		GVL.B_LengthStep := GVL.B_LengthStep + 1;
		GVL.HMI_B_RowSelectedCmd := 0;
		GVL.HMI_B_EditCmdReq := 0;

	// Insert Command Data To Step Table after line selected
	22:
		//GVL.HMI_B_SelectedStepNo := GVL.HMI_B_EditStepNo;
		FOR i := GVL.B_LengthStep TO (GVL.HMI_B_EditStepNo + 1) BY -1 DO
			GVL_1.Step_Cr_B[i+1] := GVL_1.Step_Cr_B[i];
		END_FOR
		GVL_1.Step_Cr_B[GVL.HMI_B_EditStepNo + 1].GroupCmd := 0;
		GVL_1.Step_Cr_B[GVL.HMI_B_EditStepNo + 1].Cmd := 0;
		GVL_1.Step_Cr_B[GVL.HMI_B_EditStepNo + 1].P1 := 0;
		GVL_1.Step_Cr_B[GVL.HMI_B_EditStepNo + 1].P2 := 0;
		GVL_1.Step_Cr_B[GVL.HMI_B_EditStepNo + 1].P3 := 0;
		GVL_1.Step_Cr_B[GVL.HMI_B_EditStepNo + 1].P4 := 0;
		GVL_1.Step_Cr_B[GVL.HMI_B_EditStepNo + 1].P5 := 0;
		GVL_1.Step_Cr_B[GVL.HMI_B_EditStepNo + 1].Note := '';
		GVL.B_LengthStep := GVL.B_LengthStep + 1;
		GVL.HMI_B_EditCmdReq := 0;

// 	// Delete Command Data From Step Table
// 	23:
// 		//GVL.HMI_B_SelectedStepNo := GVL.HMI_B_EditStepNo;
// 		FOR i := (GVL.HMI_B_EditStepNo) TO (GVL.B_LengthStep -1) BY 1 DO
// 			GVL_1.Step_Cr_B[i] := GVL_1.Step_Cr_B[i+1];
// 		END_FOR
// 		GVL_1.Step_Cr_B[GVL.B_LengthStep].GroupCmd := 0;
// 		GVL_1.Step_Cr_B[GVL.B_LengthStep].Cmd := 0;
// 		GVL_1.Step_Cr_B[GVL.B_LengthStep].P1 := 0;
// 		GVL_1.Step_Cr_B[GVL.B_LengthStep].P2 := 0;
// 		GVL_1.Step_Cr_B[GVL.B_LengthStep].P3 := 0;
// 		GVL_1.Step_Cr_B[GVL.B_LengthStep].P4 := 0;
// 		GVL_1.Step_Cr_B[GVL.B_LengthStep].P5 := 0;
// 		GVL_1.Step_Cr_B[GVL.B_LengthStep].Note := '';
// 		GVL.HMI_B_EditCmdReq := 0;
// 		GVL.B_LengthStep := GVL.B_LengthStep - 1;

	//============================================================
	// COPY SINGLE STEP
	// HMI_A_EditCmdReq = 25
	//============================================================
	25:
	
		IF (GVL.HMI_B_SelectedStepNo >= 1)
		   AND (GVL.HMI_B_SelectedStepNo <= GVL.B_LengthStep)
		THEN
	
			GVL.B_StepClipboard :=
				GVL_1.Step_Cr_B[GVL.HMI_B_SelectedStepNo];
	
			GVL.B_StepClipboardValid := TRUE;
	
		END_IF;
	
		GVL.HMI_B_EditCmdReq := 0;
		
	//============================================================
	// PASTE SINGLE STEP
	// Ghi đè vào step đang chọn
	//============================================================
	26:
	
		IF GVL.B_StepClipboardValid	
		   AND (GVL.HMI_B_SelectedStepNo >= 1)
		THEN
	
			GVL_1.Step_Cr_B[GVL.HMI_B_SelectedStepNo] :=
				GVL.B_StepClipboard;
	
			//----------------------------------------------------
			// Nếu paste ra ngoài LengthStep hiện tại
			//----------------------------------------------------
			IF GVL.HMI_B_SelectedStepNo > GVL.B_LengthStep THEN
				GVL.B_LengthStep := GVL.HMI_B_SelectedStepNo;
			END_IF;
	
		END_IF;
	
		GVL.HMI_B_RowSelectedCmd := 0;
		GVL.HMI_B_EditCmdReq := 0;
		
	//============================================================
	// COPY STEP BLOCK
	// HMI_A_EditCmdReq = 28
	//
	// Copy từ HMI_A_CopyStartStep đến HMI_A_CopyEndStep
	//============================================================
	28:
	
		//--------------------------------------------------------
		// Kiểm tra range hợp lệ
		//--------------------------------------------------------
		IF (GVL.HMI_B_CopyStartStep >= 1)
		   AND
		   (GVL.HMI_B_CopyEndStep >= GVL.HMI_B_CopyStartStep)
		   AND
		   (GVL.HMI_B_CopyEndStep <= GVL.B_LengthStep)
		THEN
	
			//----------------------------------------------------
			// Tính số step cần copy
			//----------------------------------------------------
			GVL.AB_StepCopyCount := GVL.HMI_B_CopyEndStep - GVL.HMI_B_CopyStartStep + 1;
	
			//----------------------------------------------------
			// Giới hạn clipboard tối đa 1000 step
			//----------------------------------------------------
			IF GVL.AB_StepCopyCount <= 1000 THEN
	
				FOR i := 1 TO GVL.AB_StepCopyCount DO
	
					GVL.AB_StepBlockClipboard[i] := GVL_1.Step_Cr_B[GVL.HMI_B_CopyStartStep + i - 1];
	
				END_FOR;
	
				//------------------------------------------------
				// Lưu range nguồn để debug / HMI
				//------------------------------------------------
				GVL.B_StepCopyStart := GVL.HMI_B_CopyStartStep;
	
				GVL.B_StepCopyEnd := GVL.HMI_B_CopyEndStep;
	
				GVL.AB_StepBlockClipboardValid := TRUE;
	
			ELSE
	
				//------------------------------------------------
				// Có thể set alarm:
				// block copy quá 100 step
				//------------------------------------------------
				GVL.AB_StepBlockClipboardValid := FALSE;
	
			END_IF;
	
		END_IF;
	
		GVL.HMI_B_EditCmdReq := 0;
		
		//============================================================
	// PASTE STEP BLOCK - INSERT MODE
	// HMI_A_EditCmdReq = 29
	//
	// Ví dụ:
	// clipboard = 5 step
	// Paste tại Step 20
	//
	// Step 20 cũ → 25
	// Step 21 cũ → 26
	// ...
	//
	// Clipboard → Step 20..24
	//============================================================
	29:
	
		IF GVL.AB_StepBlockClipboardValid
		   AND (GVL.AB_StepCopyCount > 0)
		   AND (GVL.HMI_B_SelectedStepNo >= 1)
		THEN
	
			//----------------------------------------------------
			// Kiểm tra không vượt kích thước Step_Cr_A
			//
			// Ví dụ Step_Cr_A[1..500]
			//----------------------------------------------------
			IF (GVL.B_LengthStep + GVL.AB_StepCopyCount) <= 500 THEN
	
				//------------------------------------------------
				// Dịch các step cũ xuống dưới.
				//
				// PHẢI chạy từ dưới lên để không ghi đè dữ liệu.
				//------------------------------------------------
				FOR i := GVL.B_LengthStep TO GVL.HMI_B_SelectedStepNo BY -1 DO
	
					GVL_1.Step_Cr_B[i + GVL.AB_StepCopyCount] := GVL_1.Step_Cr_B[i];
	
				END_FOR;
	
	
				//------------------------------------------------
				// Paste clipboard
				//------------------------------------------------
				FOR i := 1 TO GVL.AB_StepCopyCount DO
	
					GVL_1.Step_Cr_B[GVL.HMI_B_SelectedStepNo + i - 1] := GVL.AB_StepBlockClipboard[i];
	
				END_FOR;
	
	
				//------------------------------------------------
				// Cập nhật tổng số step
				//------------------------------------------------
				GVL.B_LengthStep := GVL.B_LengthStep + GVL.AB_StepCopyCount;
	
	
				//------------------------------------------------
				// Reset select row
				//------------------------------------------------
				GVL.HMI_B_RowSelectedCmd := 0;
	
			END_IF;
	
		END_IF;
	
		GVL.HMI_B_EditCmdReq := 0;
			
END_CASE;

// Delete Command Data From Step Table
Delete_one_Step_B(IN := GVL.HMI_B_EditCmdReq_Arr[8], PT := T#10MS);
IF Delete_one_Step_B.Q THEN
	//GVL.HMI_B_SelectedStepNo := GVL.HMI_B_EditStepNo;
	FOR i := (GVL.HMI_B_EditStepNo) TO (GVL.B_LengthStep -1) BY 1 DO
		GVL_1.Step_Cr_B[i] := GVL_1.Step_Cr_B[i+1];
	END_FOR
	GVL_1.Step_Cr_B[GVL.B_LengthStep].GroupCmd := 0;
	GVL_1.Step_Cr_B[GVL.B_LengthStep].Cmd := 0;
	GVL_1.Step_Cr_B[GVL.B_LengthStep].P1 := 0;
	GVL_1.Step_Cr_B[GVL.B_LengthStep].P2 := 0;
	GVL_1.Step_Cr_B[GVL.B_LengthStep].P3 := 0;
	GVL_1.Step_Cr_B[GVL.B_LengthStep].P4 := 0;
	GVL_1.Step_Cr_B[GVL.B_LengthStep].P5 := 0;
	GVL_1.Step_Cr_B[GVL.B_LengthStep].Note := '';
	GVL.HMI_B_EditCmdReq_Arr[8] := FALSE;
	GVL.B_LengthStep := GVL.B_LengthStep - 1;
END_IF

// Delete ALL Command Data From Step Table
Delete_all_Step_B(IN := GVL.HMI_B_EditCmdReq_Arr[9], PT := T#2S);
IF Delete_all_Step_B.Q THEN
	//GVL.HMI_B_SelectedStepNo := GVL.HMI_B_EditStepNo;
	FOR i := 0 TO (GVL.B_LengthStep) BY 1 DO
		GVL_1.Step_Cr_B[i].GroupCmd := 0;
		GVL_1.Step_Cr_B[i].Cmd := 0;
		GVL_1.Step_Cr_B[i].P1 := 0;
		GVL_1.Step_Cr_B[i].P2 := 0;
		GVL_1.Step_Cr_B[i].P3 := 0;
		GVL_1.Step_Cr_B[i].P4 := 0;
		GVL_1.Step_Cr_B[i].P5 := 0;
		GVL_1.Step_Cr_B[i].Note := '';
	END_FOR
	
	GVL.HMI_B_EditCmdReq_Arr[8] := FALSE;
	GVL.B_LengthStep := GVL.B_LengthStep - 1;
END_IF


// Enable bit chon nhom lenh
FOR i := 0 TO 10 DO
	IF (GVL.HMI_B_EditGroupCmd >= 0) AND (i = GVL.HMI_B_EditGroupCmd) THEN 
    	GVL.HMI_B_EditSelgroupCmd[i] := TRUE;
	ELSE
		GVL.HMI_B_EditSelgroupCmd[i] := FALSE;
	END_IF
END_FOR;
END_ACTION

ACTION ACT_View_Edit_Point_A:
// Chuyen doi ten diem khi lam o phan jog va teaching
IF GVL.HMI_A_ChangeSelectedPoint THEN
	GVL.HMI_A_Edit_Pos_Name := GVL_1.Point_Name_A[GVL.DW_[10]];
	GVL.HMI_A_ChangeSelectedPoint := FALSE;
END_IF

// Lua chon Cac diem can View va Edit 
CASE GVL.HMI_A_PointViewCmd OF
    1:
        GVL.HMI_A_ViewStartPoint := MAX(1, GVL.HMI_A_ViewStartPoint - 1);

    2:
        GVL.HMI_A_ViewStartPoint := MIN(491, GVL.HMI_A_ViewStartPoint + 1);

    3:
        GVL.HMI_A_ViewStartPoint := MAX(1, GVL.HMI_A_ViewStartPoint - 10);

    4:
        GVL.HMI_A_ViewStartPoint := MIN(491, GVL.HMI_A_ViewStartPoint + 10);

    5:
        GVL.HMI_A_ViewStartPoint := 1;

    6:
        GVL.HMI_A_ViewStartPoint := 491;

END_CASE;

GVL.HMI_A_PointViewCmd := 0;

// Refresh toa do hien thi tren HMI
FOR i := 1 TO 10 DO
    idx := GVL.HMI_A_ViewStartPoint + i - 1;

    GVL.HMI_A_PointNo[i]   := idx;
    GVL.HMI_A_View_Pos_Name[i] := GVL_1.Point_Name_A[idx];
    GVL.HMI_A_View_Pos_X[i]    := GVL_1.DATA_RB_A.X_POS[idx];
	GVL.HMI_A_View_Pos_Y[i]    := GVL_1.DATA_RB_A.Y_POS[idx];
	GVL.HMI_A_View_Pos_Z[i]    := GVL_1.DATA_RB_A.Z_POS[idx];
	GVL.HMI_A_View_Pos_R[i]    := GVL_1.DATA_RB_A.R_POS[idx];
END_FOR

// Tinh diem lua chon thuc te tren PLC tu HMI
//GVL.HMI_A_Poi := HMI_PointStartIndex + HMI_PointSelectedRow - 1;

// Xu ly chon dong
FOR i := 1 TO 10 DO
    IF (GVL.HMI_A_RowSelectedPoint = i) THEN
		GVL.HMI_A_RowSelectedPoint_Array[i] := TRUE;
		GVL.HMI_A_PointNoSelected := i + GVL.HMI_A_ViewStartPoint - 1;
	ELSE
		GVL.HMI_A_RowSelectedPoint_Array[i] := FALSE;
    END_IF;
END_FOR;


// Edit Point
// Load Point to Edit
IF GVL.HMI_A_EditPointReq = 20 THEN
    GVL.HMI_A_Edit_PointNo   := GVL.HMI_A_PointNoSelected;
    GVL.HMI_A_Edit_Pos_Name  := GVL_1.Point_Name_A[GVL.HMI_A_PointNoSelected];
    GVL.HMI_A_Edit_Pos_X     := GVL_1.DATA_RB_A.X_POS[GVL.HMI_A_PointNoSelected];
    GVL.HMI_A_Edit_Pos_Y     := GVL_1.DATA_RB_A.Y_POS[GVL.HMI_A_PointNoSelected];
    GVL.HMI_A_Edit_Pos_Z     := GVL_1.DATA_RB_A.Z_POS[GVL.HMI_A_PointNoSelected];
    GVL.HMI_A_Edit_Pos_R     := GVL_1.DATA_RB_A.R_POS[GVL.HMI_A_PointNoSelected];

    GVL.HMI_A_EditPointReq := 0;
END_IF

// Delete Point to Edit
Delete_one_point(IN:= GVL.HMI_A_EditPointReq_Arr[6], PT := T#2S);
// IF GVL.HMI_A_EditPointReq = 23 THEN
//     GVL.HMI_A_Edit_PointNo   := GVL.HMI_A_PointNoSelected;
//     GVL.HMI_A_Edit_Pos_Name  := '';
//     GVL.HMI_A_Edit_Pos_X     := 0;
//     GVL.HMI_A_Edit_Pos_Y     := 0;
//     GVL.HMI_A_Edit_Pos_Z     := 0;
//     GVL.HMI_A_Edit_Pos_R     := 0;
// END_IF
IF Delete_one_point.Q THEN
	IF (GVL.HMI_A_PointNoSelected >= 1) AND (GVL.HMI_A_PointNoSelected <= 500) THEN

        //----------------------------------------------------
        // Xóa dữ liệu thật
        //----------------------------------------------------
        GVL_1.Point_Name_A[GVL.HMI_A_PointNoSelected] := '';

        GVL_1.DATA_RB_A.X_POS[GVL.HMI_A_PointNoSelected] := 0.0;

        GVL_1.DATA_RB_A.Y_POS[GVL.HMI_A_PointNoSelected] := 0.0;

        GVL_1.DATA_RB_A.Z_POS[GVL.HMI_A_PointNoSelected] := 0.0;

        GVL_1.DATA_RB_A.R_POS[GVL.HMI_A_PointNoSelected] := 0.0;

	END_IF;
	GVL.HMI_A_EditPointReq := 0;
	GVL.HMI_A_EditPointReq_Arr[6] := FALSE;
END_IF

// Save Point Data
IF GVL.HMI_A_EditPointReq = 24 THEN
    GVL_1.Point_Name_A[GVL.HMI_A_PointNoSelected]      := GVL.HMI_A_Edit_Pos_Name;
    GVL_1.DATA_RB_A.X_POS[GVL.HMI_A_PointNoSelected]   := GVL.HMI_A_Edit_Pos_X;
    GVL_1.DATA_RB_A.Y_POS[GVL.HMI_A_PointNoSelected]   := GVL.HMI_A_Edit_Pos_Y;
    GVL_1.DATA_RB_A.Z_POS[GVL.HMI_A_PointNoSelected]   := GVL.HMI_A_Edit_Pos_Z;
    GVL_1.DATA_RB_A.R_POS[GVL.HMI_A_PointNoSelected]   := GVL.HMI_A_Edit_Pos_R;

    GVL.HMI_A_EditPointReq := 0;
END_IF

// Add Point to Step Table
IF GVL.HMI_A_EditPointReq = 21 THEN
    GVL.HMI_A_Edit_PointNo   := GVL.HMI_A_PointNoSelected;
    GVL.HMI_A_Edit_Pos_Name  := GVL_1.Point_Name_A[GVL.HMI_A_PointNoSelected];
    GVL.HMI_A_Edit_Pos_X     := GVL_1.DATA_RB_A.X_POS[GVL.HMI_A_PointNoSelected];
    GVL.HMI_A_Edit_Pos_Y     := GVL_1.DATA_RB_A.Y_POS[GVL.HMI_A_PointNoSelected];
    GVL.HMI_A_Edit_Pos_Z     := GVL_1.DATA_RB_A.Z_POS[GVL.HMI_A_PointNoSelected];
    GVL.HMI_A_Edit_Pos_R     := GVL_1.DATA_RB_A.R_POS[GVL.HMI_A_PointNoSelected];

    GVL.HMI_A_EditPointReq := 0;
END_IF

//============================================================
// COPY POINT
//
// HMI_A_EditPointReq = 25
//
// Copy toàn bộ dữ liệu của Point đang được chọn
// vào Clipboard.
//============================================================
IF GVL.HMI_A_EditPointReq = 25 THEN

    //--------------------------------------------------------
    // Kiểm tra PointNo hợp lệ
    // Thay 500 bằng số Point tối đa thực tế của anh
    //--------------------------------------------------------
    IF (GVL.HMI_A_PointNoSelected >= 1)
       AND (GVL.HMI_A_PointNoSelected <= 500)
    THEN

        //----------------------------------------------------
        // Lưu Point nguồn
        //----------------------------------------------------
        GVL.A_PointClipboardSourceNo := GVL.HMI_A_PointNoSelected;

        //----------------------------------------------------
        // Copy Name
        //----------------------------------------------------
        GVL.A_PointClipboardName := GVL_1.Point_Name_A[GVL.HMI_A_PointNoSelected];

        //----------------------------------------------------
        // Copy Position
        //----------------------------------------------------
        GVL.A_PointClipboardX := GVL_1.DATA_RB_A.X_POS[GVL.HMI_A_PointNoSelected];

        GVL.A_PointClipboardY := GVL_1.DATA_RB_A.Y_POS[GVL.HMI_A_PointNoSelected];

        GVL.A_PointClipboardZ := GVL_1.DATA_RB_A.Z_POS[GVL.HMI_A_PointNoSelected];

        GVL.A_PointClipboardR := GVL_1.DATA_RB_A.R_POS[GVL.HMI_A_PointNoSelected];

        //----------------------------------------------------
        // Clipboard đã có dữ liệu
        //----------------------------------------------------
        GVL.A_PointClipboardValid := TRUE;

    END_IF;

    //--------------------------------------------------------
    // Reset request
    //--------------------------------------------------------
    GVL.HMI_A_EditPointReq := 0;

END_IF;

//============================================================
// PASTE POINT
//
// HMI_A_EditPointReq = 26
//
// Paste dữ liệu Clipboard vào Point đang được chọn.
//============================================================
IF GVL.HMI_A_EditPointReq = 26 THEN

    //--------------------------------------------------------
    // Chỉ Paste khi Clipboard có dữ liệu
    //--------------------------------------------------------
    IF GVL.A_PointClipboardValid AND (GVL.HMI_A_PointNoSelected >= 1) AND (GVL.HMI_A_PointNoSelected <= 500) THEN

        //----------------------------------------------------
        // Paste Name
        //----------------------------------------------------
        GVL_1.Point_Name_A[GVL.HMI_A_PointNoSelected] := GVL.A_PointClipboardName;

        //----------------------------------------------------
        // Paste Position
        //----------------------------------------------------
        GVL_1.DATA_RB_A.X_POS[GVL.HMI_A_PointNoSelected] := GVL.A_PointClipboardX;

        GVL_1.DATA_RB_A.Y_POS[GVL.HMI_A_PointNoSelected] := GVL.A_PointClipboardY;

        GVL_1.DATA_RB_A.Z_POS[GVL.HMI_A_PointNoSelected] := GVL.A_PointClipboardZ;

        GVL_1.DATA_RB_A.R_POS[GVL.HMI_A_PointNoSelected] := GVL.A_PointClipboardR;


//         //----------------------------------------------------
//         // Đồng thời cập nhật vùng Edit để HMI hiển thị
//         // ngay dữ liệu vừa Paste
//         //----------------------------------------------------
//         GVL.HMI_A_Edit_PointNo := GVL.HMI_A_PointNoSelected;
// 
//         GVL.HMI_A_Edit_Pos_Name := GVL.A_PointClipboardName;
// 
//         GVL.HMI_A_Edit_Pos_X := GVL.A_PointClipboardX;
// 
//         GVL.HMI_A_Edit_Pos_Y := GVL.A_PointClipboardY;
// 
//         GVL.HMI_A_Edit_Pos_Z := GVL.A_PointClipboardZ;
// 
//         GVL.HMI_A_Edit_Pos_R := GVL.A_PointClipboardR;

    END_IF;

    //--------------------------------------------------------
    // Không xóa Clipboard.
    //
    // Nhờ vậy có thể:
    // Copy P10 → Paste P20 → Paste P21 → Paste P22...
    //--------------------------------------------------------

    GVL.HMI_A_EditPointReq := 0;

END_IF;

//============================================================
// DELETE ALL POINTS
//
// HMI_A_EditPointReq = 27
//
// Xóa toàn bộ Point Database.
//============================================================

Delete_all_point(IN := GVL.HMI_A_EditPointReq_Arr[7], PT := T#2S);
IF Delete_all_point.Q THEN

    FOR iPoint := 1 TO 500 DO

        //----------------------------------------------------
        // Clear Name
        //----------------------------------------------------
        GVL_1.Point_Name_A[iPoint] := '';

        //----------------------------------------------------
        // Clear Position
        //----------------------------------------------------
        GVL_1.DATA_RB_A.X_POS[iPoint] := 0.0;
        GVL_1.DATA_RB_A.Y_POS[iPoint] := 0.0;
        GVL_1.DATA_RB_A.Z_POS[iPoint] := 0.0;
        GVL_1.DATA_RB_A.R_POS[iPoint] := 0.0;

    END_FOR;


    //--------------------------------------------------------
    // Clear vùng Edit trên HMI
    //--------------------------------------------------------
    GVL.HMI_A_Edit_PointNo  := 0;
    GVL.HMI_A_Edit_Pos_Name := '';

    GVL.HMI_A_Edit_Pos_X := 0.0;
    GVL.HMI_A_Edit_Pos_Y := 0.0;
    GVL.HMI_A_Edit_Pos_Z := 0.0;
    GVL.HMI_A_Edit_Pos_R := 0.0;


    //--------------------------------------------------------
    // Reset Point đang chọn
    //--------------------------------------------------------
    GVL.HMI_A_PointNoSelected := 0;


    //--------------------------------------------------------
    // Em khuyên KHÔNG xóa Clipboard.
    //
    // Nếu Delete All nhầm, dữ liệu Point vừa Copy vẫn còn
    // và có thể Paste lại.
    //--------------------------------------------------------

    GVL.HMI_A_EditPointReq := 0;
	GVL.HMI_A_EditPointReq_Arr[7] := FALSE;

END_IF;
END_ACTION

ACTION ACT_View_Edit_Point_B:
// ============================================================
// CREATE ACTION: ACT_View_Edit_Point_B
// Parent POU: POU_HMI_CONTROL_ROBOT
// Source mirrored from: ACT_View_Edit_Point_A
// ============================================================

// Chuyen doi ten diem khi lam o phan jog va teaching
IF GVL.HMI_B_ChangeSelectedPoint THEN
	GVL.HMI_B_Edit_Pos_Name := GVL_1.Point_Name_B[GVL.DW_[12]];
	GVL.HMI_B_ChangeSelectedPoint := FALSE;
END_IF

// Lua chon Cac diem can View va Edit 
CASE GVL.HMI_B_PointViewCmd OF
    1:
        GVL.HMI_B_ViewStartPoint := MAX(1, GVL.HMI_B_ViewStartPoint - 1);

    2:
        GVL.HMI_B_ViewStartPoint := MIN(491, GVL.HMI_B_ViewStartPoint + 1);

    3:
        GVL.HMI_B_ViewStartPoint := MAX(1, GVL.HMI_B_ViewStartPoint - 10);

    4:
        GVL.HMI_B_ViewStartPoint := MIN(491, GVL.HMI_B_ViewStartPoint + 10);

    5:
        GVL.HMI_B_ViewStartPoint := 1;

    6:
        GVL.HMI_B_ViewStartPoint := 491;

END_CASE;

GVL.HMI_B_PointViewCmd := 0;

// Refresh toa do hien thi tren HMI
FOR i := 1 TO 10 DO
    idx := GVL.HMI_B_ViewStartPoint + i - 1;

    GVL.HMI_B_PointNo[i]   := idx;
    GVL.HMI_B_View_Pos_Name[i] := GVL_1.Point_Name_B[idx];
    GVL.HMI_B_View_Pos_X[i]    := GVL_1.DATA_RB_B.X_POS[idx];
	GVL.HMI_B_View_Pos_Y[i]    := GVL_1.DATA_RB_B.Y_POS[idx];
	GVL.HMI_B_View_Pos_Z[i]    := GVL_1.DATA_RB_B.Z_POS[idx];
	GVL.HMI_B_View_Pos_R[i]    := GVL_1.DATA_RB_B.R_POS[idx];
END_FOR

// Tinh diem lua chon thuc te tren PLC tu HMI
//GVL.HMI_B_Poi := HMI_PointStartIndex + HMI_PointSelectedRow - 1;

// Xu ly chon dong
FOR i := 1 TO 10 DO
    IF (GVL.HMI_B_RowSelectedPoint = i) THEN
		GVL.HMI_B_RowSelectedPoint_Array[i] := TRUE;
		GVL.HMI_B_PointNoSelected := i + GVL.HMI_B_ViewStartPoint - 1;
	ELSE
		GVL.HMI_B_RowSelectedPoint_Array[i] := FALSE;
    END_IF;
END_FOR;


// Edit Point
// Load Point to Edit
IF GVL.HMI_B_EditPointReq = 20 THEN
    GVL.HMI_B_Edit_PointNo   := GVL.HMI_B_PointNoSelected;
    GVL.HMI_B_Edit_Pos_Name  := GVL_1.Point_Name_B[GVL.HMI_B_PointNoSelected];
    GVL.HMI_B_Edit_Pos_X     := GVL_1.DATA_RB_B.X_POS[GVL.HMI_B_PointNoSelected];
    GVL.HMI_B_Edit_Pos_Y     := GVL_1.DATA_RB_B.Y_POS[GVL.HMI_B_PointNoSelected];
    GVL.HMI_B_Edit_Pos_Z     := GVL_1.DATA_RB_B.Z_POS[GVL.HMI_B_PointNoSelected];
    GVL.HMI_B_Edit_Pos_R     := GVL_1.DATA_RB_B.R_POS[GVL.HMI_B_PointNoSelected];

    GVL.HMI_B_EditPointReq := 0;
END_IF

// Delete Point to Edit
Delete_one_point_B(IN:= GVL.HMI_B_EditPointReq_Arr[6], PT := T#2S);
// IF GVL.HMI_B_EditPointReq = 23 THEN
//     GVL.HMI_B_Edit_PointNo   := GVL.HMI_B_PointNoSelected;
//     GVL.HMI_B_Edit_Pos_Name  := '';
//     GVL.HMI_B_Edit_Pos_X     := 0;
//     GVL.HMI_B_Edit_Pos_Y     := 0;
//     GVL.HMI_B_Edit_Pos_Z     := 0;
//     GVL.HMI_B_Edit_Pos_R     := 0;
// END_IF
IF Delete_one_point_B.Q THEN
	IF (GVL.HMI_B_PointNoSelected >= 1) AND (GVL.HMI_B_PointNoSelected <= 500) THEN

        //----------------------------------------------------
        // Xóa dữ liệu thật
        //----------------------------------------------------
        GVL_1.Point_Name_B[GVL.HMI_B_PointNoSelected] := '';

        GVL_1.DATA_RB_B.X_POS[GVL.HMI_B_PointNoSelected] := 0.0;

        GVL_1.DATA_RB_B.Y_POS[GVL.HMI_B_PointNoSelected] := 0.0;

        GVL_1.DATA_RB_B.Z_POS[GVL.HMI_B_PointNoSelected] := 0.0;

        GVL_1.DATA_RB_B.R_POS[GVL.HMI_B_PointNoSelected] := 0.0;

	END_IF;
	GVL.HMI_B_EditPointReq := 0;
	GVL.HMI_B_EditPointReq_Arr[6] := FALSE;
END_IF

// Save Point Data
IF GVL.HMI_B_EditPointReq = 24 THEN
    GVL_1.Point_Name_B[GVL.HMI_B_PointNoSelected]      := GVL.HMI_B_Edit_Pos_Name;
    GVL_1.DATA_RB_B.X_POS[GVL.HMI_B_PointNoSelected]   := GVL.HMI_B_Edit_Pos_X;
    GVL_1.DATA_RB_B.Y_POS[GVL.HMI_B_PointNoSelected]   := GVL.HMI_B_Edit_Pos_Y;
    GVL_1.DATA_RB_B.Z_POS[GVL.HMI_B_PointNoSelected]   := GVL.HMI_B_Edit_Pos_Z;
    GVL_1.DATA_RB_B.R_POS[GVL.HMI_B_PointNoSelected]   := GVL.HMI_B_Edit_Pos_R;

    GVL.HMI_B_EditPointReq := 0;
END_IF

// Add Point to Step Table
IF GVL.HMI_B_EditPointReq = 21 THEN
    GVL.HMI_B_Edit_PointNo   := GVL.HMI_B_PointNoSelected;
    GVL.HMI_B_Edit_Pos_Name  := GVL_1.Point_Name_B[GVL.HMI_B_PointNoSelected];
    GVL.HMI_B_Edit_Pos_X     := GVL_1.DATA_RB_B.X_POS[GVL.HMI_B_PointNoSelected];
    GVL.HMI_B_Edit_Pos_Y     := GVL_1.DATA_RB_B.Y_POS[GVL.HMI_B_PointNoSelected];
    GVL.HMI_B_Edit_Pos_Z     := GVL_1.DATA_RB_B.Z_POS[GVL.HMI_B_PointNoSelected];
    GVL.HMI_B_Edit_Pos_R     := GVL_1.DATA_RB_B.R_POS[GVL.HMI_B_PointNoSelected];

    GVL.HMI_B_EditPointReq := 0;
END_IF

//============================================================
// COPY POINT
//
// HMI_A_EditPointReq = 25
//
// Copy toàn bộ dữ liệu của Point đang được chọn
// vào Clipboard.
//============================================================
IF GVL.HMI_B_EditPointReq = 25 THEN

    //--------------------------------------------------------
    // Kiểm tra PointNo hợp lệ
    // Thay 500 bằng số Point tối đa thực tế của anh
    //--------------------------------------------------------
    IF (GVL.HMI_B_PointNoSelected >= 1)
       AND (GVL.HMI_B_PointNoSelected <= 500)
    THEN

        //----------------------------------------------------
        // Lưu Point nguồn
        //----------------------------------------------------
        GVL.B_PointClipboardSourceNo := GVL.HMI_B_PointNoSelected;

        //----------------------------------------------------
        // Copy Name
        //----------------------------------------------------
        GVL.B_PointClipboardName := GVL_1.Point_Name_B[GVL.HMI_B_PointNoSelected];

        //----------------------------------------------------
        // Copy Position
        //----------------------------------------------------
        GVL.B_PointClipboardX := GVL_1.DATA_RB_B.X_POS[GVL.HMI_B_PointNoSelected];

        GVL.B_PointClipboardY := GVL_1.DATA_RB_B.Y_POS[GVL.HMI_B_PointNoSelected];

        GVL.B_PointClipboardZ := GVL_1.DATA_RB_B.Z_POS[GVL.HMI_B_PointNoSelected];

        GVL.B_PointClipboardR := GVL_1.DATA_RB_B.R_POS[GVL.HMI_B_PointNoSelected];

        //----------------------------------------------------
        // Clipboard đã có dữ liệu
        //----------------------------------------------------
        GVL.B_PointClipboardValid := TRUE;

    END_IF;

    //--------------------------------------------------------
    // Reset request
    //--------------------------------------------------------
    GVL.HMI_B_EditPointReq := 0;

END_IF;

//============================================================
// PASTE POINT
//
// HMI_A_EditPointReq = 26
//
// Paste dữ liệu Clipboard vào Point đang được chọn.
//============================================================
IF GVL.HMI_B_EditPointReq = 26 THEN

    //--------------------------------------------------------
    // Chỉ Paste khi Clipboard có dữ liệu
    //--------------------------------------------------------
    IF GVL.B_PointClipboardValid AND (GVL.HMI_B_PointNoSelected >= 1) AND (GVL.HMI_B_PointNoSelected <= 500) THEN

        //----------------------------------------------------
        // Paste Name
        //----------------------------------------------------
        GVL_1.Point_Name_B[GVL.HMI_B_PointNoSelected] := GVL.B_PointClipboardName;

